aff1Ge[0  , 0] := 1.00000E+01; aff1Ge[0  , 1] := -2.69562E+01;
aff1Ge[1  , 0] := 1.99800E+01; aff1Ge[1  , 1] := -2.74605E+01;
aff1Ge[2  , 0] := 2.99600E+01; aff1Ge[2  , 1] := -2.88439E+01;
aff1Ge[3  , 0] := 3.99400E+01; aff1Ge[3  , 1] := -2.93110E+01;
aff1Ge[4  , 0] := 4.99200E+01; aff1Ge[4  , 1] := -2.98763E+01;
aff1Ge[5  , 0] := 5.99000E+01; aff1Ge[5  , 1] := -3.00073E+01;
aff1Ge[6  , 0] := 6.98800E+01; aff1Ge[6  , 1] := -2.96407E+01;
aff1Ge[7  , 0] := 7.98600E+01; aff1Ge[7  , 1] := -2.88592E+01;
aff1Ge[8  , 0] := 8.98400E+01; aff1Ge[8  , 1] := -2.77849E+01;
aff1Ge[9  , 0] := 9.98200E+01; aff1Ge[9  , 1] := -2.65823E+01;
aff1Ge[10 , 0] := 1.09800E+02; aff1Ge[10 , 1] := -2.53647E+01;
aff1Ge[11 , 0] := 1.19780E+02; aff1Ge[11 , 1] := -2.42993E+01;
aff1Ge[12 , 0] := 1.29760E+02; aff1Ge[12 , 1] := -2.30319E+01;
aff1Ge[13 , 0] := 1.39740E+02; aff1Ge[13 , 1] := -2.17280E+01;
aff1Ge[14 , 0] := 1.49720E+02; aff1Ge[14 , 1] := -2.05826E+01;
aff1Ge[15 , 0] := 1.59700E+02; aff1Ge[15 , 1] := -1.95740E+01;
aff1Ge[16 , 0] := 1.69680E+02; aff1Ge[16 , 1] := -1.87194E+01;
aff1Ge[17 , 0] := 1.79660E+02; aff1Ge[17 , 1] := -1.81208E+01;
aff1Ge[18 , 0] := 1.89640E+02; aff1Ge[18 , 1] := -1.70898E+01;
aff1Ge[19 , 0] := 1.99620E+02; aff1Ge[19 , 1] := -1.62563E+01;
aff1Ge[20 , 0] := 2.09600E+02; aff1Ge[20 , 1] := -1.55355E+01;
aff1Ge[21 , 0] := 2.19580E+02; aff1Ge[21 , 1] := -1.48945E+01;
aff1Ge[22 , 0] := 2.29560E+02; aff1Ge[22 , 1] := -1.43191E+01;
aff1Ge[23 , 0] := 2.39540E+02; aff1Ge[23 , 1] := -1.37997E+01;
aff1Ge[24 , 0] := 2.49520E+02; aff1Ge[24 , 1] := -1.33294E+01;
aff1Ge[25 , 0] := 2.59500E+02; aff1Ge[25 , 1] := -1.29022E+01;
aff1Ge[26 , 0] := 2.69480E+02; aff1Ge[26 , 1] := -1.25135E+01;
aff1Ge[27 , 0] := 2.79460E+02; aff1Ge[27 , 1] := -1.21589E+01;
aff1Ge[28 , 0] := 2.89440E+02; aff1Ge[28 , 1] := -1.18350E+01;
aff1Ge[29 , 0] := 2.99420E+02; aff1Ge[29 , 1] := -1.15386E+01;
aff1Ge[30 , 0] := 3.09400E+02; aff1Ge[30 , 1] := -1.12669E+01;
aff1Ge[31 , 0] := 3.19380E+02; aff1Ge[31 , 1] := -1.10176E+01;
aff1Ge[32 , 0] := 3.29360E+02; aff1Ge[32 , 1] := -1.07885E+01;
aff1Ge[33 , 0] := 3.39340E+02; aff1Ge[33 , 1] := -1.05777E+01;
aff1Ge[34 , 0] := 3.49320E+02; aff1Ge[34 , 1] := -1.03835E+01;
aff1Ge[35 , 0] := 3.59300E+02; aff1Ge[35 , 1] := -1.02046E+01;
aff1Ge[36 , 0] := 3.69280E+02; aff1Ge[36 , 1] := -1.00390E+01;
aff1Ge[37 , 0] := 3.79260E+02; aff1Ge[37 , 1] := -9.88636E+00;
aff1Ge[38 , 0] := 3.89240E+02; aff1Ge[38 , 1] := -9.74811E+00;
aff1Ge[39 , 0] := 3.99220E+02; aff1Ge[39 , 1] := -9.61794E+00;
aff1Ge[40 , 0] := 4.09200E+02; aff1Ge[40 , 1] := -9.49749E+00;
aff1Ge[41 , 0] := 4.19180E+02; aff1Ge[41 , 1] := -9.38606E+00;
aff1Ge[42 , 0] := 4.29160E+02; aff1Ge[42 , 1] := -9.28294E+00;
aff1Ge[43 , 0] := 4.39140E+02; aff1Ge[43 , 1] := -9.18748E+00;
aff1Ge[44 , 0] := 4.49120E+02; aff1Ge[44 , 1] := -9.09912E+00;
aff1Ge[45 , 0] := 4.59100E+02; aff1Ge[45 , 1] := -9.01731E+00;
aff1Ge[46 , 0] := 4.69080E+02; aff1Ge[46 , 1] := -8.94156E+00;
aff1Ge[47 , 0] := 4.79060E+02; aff1Ge[47 , 1] := -8.87141E+00;
aff1Ge[48 , 0] := 4.89040E+02; aff1Ge[48 , 1] := -8.80645E+00;
aff1Ge[49 , 0] := 4.99020E+02; aff1Ge[49 , 1] := -8.74631E+00;
aff1Ge[50 , 0] := 5.09000E+02; aff1Ge[50 , 1] := -8.69071E+00;
aff1Ge[51 , 0] := 5.18980E+02; aff1Ge[51 , 1] := -8.63934E+00;
aff1Ge[52 , 0] := 5.28960E+02; aff1Ge[52 , 1] := -8.59192E+00;
aff1Ge[53 , 0] := 5.38940E+02; aff1Ge[53 , 1] := -8.54809E+00;
aff1Ge[54 , 0] := 5.48920E+02; aff1Ge[54 , 1] := -8.50710E+00;
aff1Ge[55 , 0] := 5.58900E+02; aff1Ge[55 , 1] := -8.47410E+00;
aff1Ge[56 , 0] := 5.68880E+02; aff1Ge[56 , 1] := -8.44688E+00;
aff1Ge[57 , 0] := 5.78860E+02; aff1Ge[57 , 1] := -8.42499E+00;
aff1Ge[58 , 0] := 5.88840E+02; aff1Ge[58 , 1] := -8.40804E+00;
aff1Ge[59 , 0] := 5.98820E+02; aff1Ge[59 , 1] := -8.39568E+00;
aff1Ge[60 , 0] := 6.08800E+02; aff1Ge[60 , 1] := -8.38763E+00;
aff1Ge[61 , 0] := 6.18780E+02; aff1Ge[61 , 1] := -8.38361E+00;
aff1Ge[62 , 0] := 6.28760E+02; aff1Ge[62 , 1] := -8.38341E+00;
aff1Ge[63 , 0] := 6.38740E+02; aff1Ge[63 , 1] := -8.38682E+00;
aff1Ge[64 , 0] := 6.48720E+02; aff1Ge[64 , 1] := -8.39368E+00;
aff1Ge[65 , 0] := 6.58700E+02; aff1Ge[65 , 1] := -8.40382E+00;
aff1Ge[66 , 0] := 6.68680E+02; aff1Ge[66 , 1] := -8.41712E+00;
aff1Ge[67 , 0] := 6.78660E+02; aff1Ge[67 , 1] := -8.43346E+00;
aff1Ge[68 , 0] := 6.88640E+02; aff1Ge[68 , 1] := -8.45275E+00;
aff1Ge[69 , 0] := 6.98620E+02; aff1Ge[69 , 1] := -8.47490E+00;
aff1Ge[70 , 0] := 7.08600E+02; aff1Ge[70 , 1] := -8.49984E+00;
aff1Ge[71 , 0] := 7.18580E+02; aff1Ge[71 , 1] := -8.52752E+00;
aff1Ge[72 , 0] := 7.28560E+02; aff1Ge[72 , 1] := -8.55788E+00;
aff1Ge[73 , 0] := 7.38540E+02; aff1Ge[73 , 1] := -8.59091E+00;
aff1Ge[74 , 0] := 7.48520E+02; aff1Ge[74 , 1] := -8.62657E+00;
aff1Ge[75 , 0] := 7.58500E+02; aff1Ge[75 , 1] := -8.66487E+00;
aff1Ge[76 , 0] := 7.68480E+02; aff1Ge[76 , 1] := -8.70579E+00;
aff1Ge[77 , 0] := 7.78460E+02; aff1Ge[77 , 1] := -8.74937E+00;
aff1Ge[78 , 0] := 7.88440E+02; aff1Ge[78 , 1] := -8.79560E+00;
aff1Ge[79 , 0] := 7.98420E+02; aff1Ge[79 , 1] := -8.84453E+00;
aff1Ge[80 , 0] := 8.08400E+02; aff1Ge[80 , 1] := -8.89620E+00;
aff1Ge[81 , 0] := 8.18380E+02; aff1Ge[81 , 1] := -8.95066E+00;
aff1Ge[82 , 0] := 8.28360E+02; aff1Ge[82 , 1] := -9.00798E+00;
aff1Ge[83 , 0] := 8.38340E+02; aff1Ge[83 , 1] := -9.06823E+00;
aff1Ge[84 , 0] := 8.48320E+02; aff1Ge[84 , 1] := -9.13150E+00;
aff1Ge[85 , 0] := 8.58300E+02; aff1Ge[85 , 1] := -9.19789E+00;
aff1Ge[86 , 0] := 8.68280E+02; aff1Ge[86 , 1] := -9.26753E+00;
aff1Ge[87 , 0] := 8.78260E+02; aff1Ge[87 , 1] := -9.34054E+00;
aff1Ge[88 , 0] := 8.88240E+02; aff1Ge[88 , 1] := -9.41707E+00;
aff1Ge[89 , 0] := 8.98220E+02; aff1Ge[89 , 1] := -9.49731E+00;
aff1Ge[90 , 0] := 9.08200E+02; aff1Ge[90 , 1] := -9.58142E+00;
aff1Ge[91 , 0] := 9.18180E+02; aff1Ge[91 , 1] := -9.66964E+00;
aff1Ge[92 , 0] := 9.28160E+02; aff1Ge[92 , 1] := -9.76220E+00;
aff1Ge[93 , 0] := 9.38140E+02; aff1Ge[93 , 1] := -9.85936E+00;
aff1Ge[94 , 0] := 9.48120E+02; aff1Ge[94 , 1] := -9.96144E+00;
aff1Ge[95 , 0] := 9.58100E+02; aff1Ge[95 , 1] := -1.00688E+01;
aff1Ge[96 , 0] := 9.68080E+02; aff1Ge[96 , 1] := -1.01817E+01;
aff1Ge[97 , 0] := 9.78060E+02; aff1Ge[97 , 1] := -1.03008E+01;
aff1Ge[98 , 0] := 9.88040E+02; aff1Ge[98 , 1] := -1.04264E+01;
aff1Ge[99 , 0] := 9.98020E+02; aff1Ge[99 , 1] := -1.05588E+01;
aff1Ge[100, 0] := 1.00800E+03; aff1Ge[100, 1] := -1.06740E+01;
aff1Ge[101, 0] := 1.01798E+03; aff1Ge[101, 1] := -1.08082E+01;
aff1Ge[102, 0] := 1.02796E+03; aff1Ge[102, 1] := -1.09580E+01;
aff1Ge[103, 0] := 1.03794E+03; aff1Ge[103, 1] := -1.11214E+01;
aff1Ge[104, 0] := 1.04792E+03; aff1Ge[104, 1] := -1.12984E+01;
aff1Ge[105, 0] := 1.05790E+03; aff1Ge[105, 1] := -1.14900E+01;
aff1Ge[106, 0] := 1.06788E+03; aff1Ge[106, 1] := -1.16973E+01;
aff1Ge[107, 0] := 1.07786E+03; aff1Ge[107, 1] := -1.19223E+01;
aff1Ge[108, 0] := 1.08784E+03; aff1Ge[108, 1] := -1.21671E+01;
aff1Ge[109, 0] := 1.09782E+03; aff1Ge[109, 1] := -1.24347E+01;
aff1Ge[110, 0] := 1.10780E+03; aff1Ge[110, 1] := -1.27288E+01;
aff1Ge[111, 0] := 1.11778E+03; aff1Ge[111, 1] := -1.30542E+01;
aff1Ge[112, 0] := 1.12776E+03; aff1Ge[112, 1] := -1.34172E+01;
aff1Ge[113, 0] := 1.13774E+03; aff1Ge[113, 1] := -1.38264E+01;
aff1Ge[114, 0] := 1.14772E+03; aff1Ge[114, 1] := -1.42937E+01;
aff1Ge[115, 0] := 1.15770E+03; aff1Ge[115, 1] := -1.48367E+01;
aff1Ge[116, 0] := 1.16768E+03; aff1Ge[116, 1] := -1.54822E+01;
aff1Ge[117, 0] := 1.17766E+03; aff1Ge[117, 1] := -1.62764E+01;
aff1Ge[118, 0] := 1.18764E+03; aff1Ge[118, 1] := -1.73070E+01;
aff1Ge[119, 0] := 1.19762E+03; aff1Ge[119, 1] := -1.87288E+01;
aff1Ge[120, 0] := 1.20760E+03; aff1Ge[120, 1] := -2.12100E+01;
aff1Ge[121, 0] := 1.21758E+03; aff1Ge[121, 1] := -2.83958E+01;
aff1Ge[122, 0] := 1.22756E+03; aff1Ge[122, 1] := -2.14204E+01;
aff1Ge[123, 0] := 1.23754E+03; aff1Ge[123, 1] := -2.02584E+01;
aff1Ge[124, 0] := 1.24752E+03; aff1Ge[124, 1] := -2.36131E+01;
aff1Ge[125, 0] := 1.25750E+03; aff1Ge[125, 1] := -1.80663E+01;
aff1Ge[126, 0] := 1.26748E+03; aff1Ge[126, 1] := -1.62455E+01;
aff1Ge[127, 0] := 1.27746E+03; aff1Ge[127, 1] := -1.49931E+01;
aff1Ge[128, 0] := 1.28744E+03; aff1Ge[128, 1] := -1.40188E+01;
aff1Ge[129, 0] := 1.29742E+03; aff1Ge[129, 1] := -1.32303E+01;
aff1Ge[130, 0] := 1.30740E+03; aff1Ge[130, 1] := -1.25660E+01;
aff1Ge[131, 0] := 1.31738E+03; aff1Ge[131, 1] := -1.19953E+01;
aff1Ge[132, 0] := 1.32736E+03; aff1Ge[132, 1] := -1.15004E+01;
aff1Ge[133, 0] := 1.33734E+03; aff1Ge[133, 1] := -1.10692E+01;
aff1Ge[134, 0] := 1.34732E+03; aff1Ge[134, 1] := -1.06941E+01;
aff1Ge[135, 0] := 1.35730E+03; aff1Ge[135, 1] := -1.03708E+01;
aff1Ge[136, 0] := 1.36728E+03; aff1Ge[136, 1] := -1.00987E+01;
aff1Ge[137, 0] := 1.37726E+03; aff1Ge[137, 1] := -9.88117E+00;
aff1Ge[138, 0] := 1.38724E+03; aff1Ge[138, 1] := -9.72484E+00;
aff1Ge[139, 0] := 1.39722E+03; aff1Ge[139, 1] := -9.66231E+00;
aff1Ge[140, 0] := 1.40720E+03; aff1Ge[140, 1] := -9.90064E+00;
aff1Ge[141, 0] := 1.41718E+03; aff1Ge[141, 1] := -9.89144E+00;
aff1Ge[142, 0] := 1.42716E+03; aff1Ge[142, 1] := -9.04354E+00;
aff1Ge[143, 0] := 1.43714E+03; aff1Ge[143, 1] := -8.44440E+00;
aff1Ge[144, 0] := 1.44712E+03; aff1Ge[144, 1] := -8.04837E+00;
aff1Ge[145, 0] := 1.45710E+03; aff1Ge[145, 1] := -7.66433E+00;
aff1Ge[146, 0] := 1.46708E+03; aff1Ge[146, 1] := -7.33565E+00;
aff1Ge[147, 0] := 1.47706E+03; aff1Ge[147, 1] := -7.03836E+00;
aff1Ge[148, 0] := 1.48704E+03; aff1Ge[148, 1] := -6.76578E+00;
aff1Ge[149, 0] := 1.49702E+03; aff1Ge[149, 1] := -6.51318E+00;
aff1Ge[150, 0] := 1.50700E+03; aff1Ge[150, 1] := -6.27757E+00;
aff1Ge[151, 0] := 1.51698E+03; aff1Ge[151, 1] := -6.05663E+00;
aff1Ge[152, 0] := 1.52696E+03; aff1Ge[152, 1] := -5.84846E+00;
aff1Ge[153, 0] := 1.53694E+03; aff1Ge[153, 1] := -5.65164E+00;
aff1Ge[154, 0] := 1.54692E+03; aff1Ge[154, 1] := -5.46502E+00;
aff1Ge[155, 0] := 1.55690E+03; aff1Ge[155, 1] := -5.28758E+00;
aff1Ge[156, 0] := 1.56688E+03; aff1Ge[156, 1] := -5.11849E+00;
aff1Ge[157, 0] := 1.57686E+03; aff1Ge[157, 1] := -4.95701E+00;
aff1Ge[158, 0] := 1.58684E+03; aff1Ge[158, 1] := -4.80260E+00;
aff1Ge[159, 0] := 1.59682E+03; aff1Ge[159, 1] := -4.65490E+00;
aff1Ge[160, 0] := 1.60680E+03; aff1Ge[160, 1] := -4.51353E+00;
aff1Ge[161, 0] := 1.61678E+03; aff1Ge[161, 1] := -4.37793E+00;
aff1Ge[162, 0] := 1.62676E+03; aff1Ge[162, 1] := -4.24779E+00;
aff1Ge[163, 0] := 1.63674E+03; aff1Ge[163, 1] := -4.12289E+00;
aff1Ge[164, 0] := 1.64672E+03; aff1Ge[164, 1] := -4.00290E+00;
aff1Ge[165, 0] := 1.65670E+03; aff1Ge[165, 1] := -3.88754E+00;
aff1Ge[166, 0] := 1.66668E+03; aff1Ge[166, 1] := -3.77652E+00;
aff1Ge[167, 0] := 1.67666E+03; aff1Ge[167, 1] := -3.66960E+00;
aff1Ge[168, 0] := 1.68664E+03; aff1Ge[168, 1] := -3.56654E+00;
aff1Ge[169, 0] := 1.69662E+03; aff1Ge[169, 1] := -3.46715E+00;
aff1Ge[170, 0] := 1.70660E+03; aff1Ge[170, 1] := -3.37123E+00;
aff1Ge[171, 0] := 1.71658E+03; aff1Ge[171, 1] := -3.27860E+00;
aff1Ge[172, 0] := 1.72656E+03; aff1Ge[172, 1] := -3.18910E+00;
aff1Ge[173, 0] := 1.73654E+03; aff1Ge[173, 1] := -3.10258E+00;
aff1Ge[174, 0] := 1.74652E+03; aff1Ge[174, 1] := -3.01889E+00;
aff1Ge[175, 0] := 1.75650E+03; aff1Ge[175, 1] := -2.93789E+00;
aff1Ge[176, 0] := 1.76648E+03; aff1Ge[176, 1] := -2.85946E+00;
aff1Ge[177, 0] := 1.77646E+03; aff1Ge[177, 1] := -2.78347E+00;
aff1Ge[178, 0] := 1.78644E+03; aff1Ge[178, 1] := -2.70981E+00;
aff1Ge[179, 0] := 1.79642E+03; aff1Ge[179, 1] := -2.63837E+00;
aff1Ge[180, 0] := 1.80640E+03; aff1Ge[180, 1] := -2.56904E+00;
aff1Ge[181, 0] := 1.81638E+03; aff1Ge[181, 1] := -2.50168E+00;
aff1Ge[182, 0] := 1.82636E+03; aff1Ge[182, 1] := -2.43620E+00;
aff1Ge[183, 0] := 1.83634E+03; aff1Ge[183, 1] := -2.37250E+00;
aff1Ge[184, 0] := 1.84632E+03; aff1Ge[184, 1] := -2.31060E+00;
aff1Ge[185, 0] := 1.85630E+03; aff1Ge[185, 1] := -2.25066E+00;
aff1Ge[186, 0] := 1.86628E+03; aff1Ge[186, 1] := -2.19265E+00;
aff1Ge[187, 0] := 1.87626E+03; aff1Ge[187, 1] := -2.13640E+00;
aff1Ge[188, 0] := 1.88624E+03; aff1Ge[188, 1] := -2.08183E+00;
aff1Ge[189, 0] := 1.89622E+03; aff1Ge[189, 1] := -2.02888E+00;
aff1Ge[190, 0] := 1.90620E+03; aff1Ge[190, 1] := -1.97748E+00;
aff1Ge[191, 0] := 1.91618E+03; aff1Ge[191, 1] := -1.92757E+00;
aff1Ge[192, 0] := 1.92616E+03; aff1Ge[192, 1] := -1.87908E+00;
aff1Ge[193, 0] := 1.93614E+03; aff1Ge[193, 1] := -1.83197E+00;
aff1Ge[194, 0] := 1.94612E+03; aff1Ge[194, 1] := -1.78618E+00;
aff1Ge[195, 0] := 1.95610E+03; aff1Ge[195, 1] := -1.74166E+00;
aff1Ge[196, 0] := 1.96608E+03; aff1Ge[196, 1] := -1.69837E+00;
aff1Ge[197, 0] := 1.97606E+03; aff1Ge[197, 1] := -1.65627E+00;
aff1Ge[198, 0] := 1.98604E+03; aff1Ge[198, 1] := -1.61531E+00;
aff1Ge[199, 0] := 1.99602E+03; aff1Ge[199, 1] := -1.57545E+00;
aff1Ge[200, 0] := 2.00600E+03; aff1Ge[200, 1] := -1.53666E+00;
aff1Ge[201, 0] := 2.01598E+03; aff1Ge[201, 1] := -1.49890E+00;
aff1Ge[202, 0] := 2.02596E+03; aff1Ge[202, 1] := -1.46214E+00;
aff1Ge[203, 0] := 2.03594E+03; aff1Ge[203, 1] := -1.42634E+00;
aff1Ge[204, 0] := 2.04592E+03; aff1Ge[204, 1] := -1.39147E+00;
aff1Ge[205, 0] := 2.05590E+03; aff1Ge[205, 1] := -1.35750E+00;
aff1Ge[206, 0] := 2.06588E+03; aff1Ge[206, 1] := -1.32440E+00;
aff1Ge[207, 0] := 2.07586E+03; aff1Ge[207, 1] := -1.29215E+00;
aff1Ge[208, 0] := 2.08584E+03; aff1Ge[208, 1] := -1.26072E+00;
aff1Ge[209, 0] := 2.09582E+03; aff1Ge[209, 1] := -1.23008E+00;
aff1Ge[210, 0] := 2.10580E+03; aff1Ge[210, 1] := -1.20020E+00;
aff1Ge[211, 0] := 2.11578E+03; aff1Ge[211, 1] := -1.17107E+00;
aff1Ge[212, 0] := 2.12576E+03; aff1Ge[212, 1] := -1.14266E+00;
aff1Ge[213, 0] := 2.13574E+03; aff1Ge[213, 1] := -1.11495E+00;
aff1Ge[214, 0] := 2.14572E+03; aff1Ge[214, 1] := -1.08791E+00;
aff1Ge[215, 0] := 2.15570E+03; aff1Ge[215, 1] := -1.06153E+00;
aff1Ge[216, 0] := 2.16568E+03; aff1Ge[216, 1] := -1.03578E+00;
aff1Ge[217, 0] := 2.17566E+03; aff1Ge[217, 1] := -1.01065E+00;
aff1Ge[218, 0] := 2.18564E+03; aff1Ge[218, 1] := -9.86115E-01;
aff1Ge[219, 0] := 2.19562E+03; aff1Ge[219, 1] := -9.62161E-01;
aff1Ge[220, 0] := 2.20560E+03; aff1Ge[220, 1] := -9.38768E-01;
aff1Ge[221, 0] := 2.21558E+03; aff1Ge[221, 1] := -9.15920E-01;
aff1Ge[222, 0] := 2.22556E+03; aff1Ge[222, 1] := -8.93600E-01;
aff1Ge[223, 0] := 2.23554E+03; aff1Ge[223, 1] := -8.71792E-01;
aff1Ge[224, 0] := 2.24552E+03; aff1Ge[224, 1] := -8.50481E-01;
aff1Ge[225, 0] := 2.25550E+03; aff1Ge[225, 1] := -8.29650E-01;
aff1Ge[226, 0] := 2.26548E+03; aff1Ge[226, 1] := -8.09280E-01;
aff1Ge[227, 0] := 2.27546E+03; aff1Ge[227, 1] := -7.89365E-01;
aff1Ge[228, 0] := 2.28544E+03; aff1Ge[228, 1] := -7.69901E-01;
aff1Ge[229, 0] := 2.29542E+03; aff1Ge[229, 1] := -7.50878E-01;
aff1Ge[230, 0] := 2.30540E+03; aff1Ge[230, 1] := -7.32285E-01;
aff1Ge[231, 0] := 2.31538E+03; aff1Ge[231, 1] := -7.14109E-01;
aff1Ge[232, 0] := 2.32536E+03; aff1Ge[232, 1] := -6.96337E-01;
aff1Ge[233, 0] := 2.33534E+03; aff1Ge[233, 1] := -6.78955E-01;
aff1Ge[234, 0] := 2.34532E+03; aff1Ge[234, 1] := -6.61952E-01;
aff1Ge[235, 0] := 2.35530E+03; aff1Ge[235, 1] := -6.45314E-01;
aff1Ge[236, 0] := 2.36528E+03; aff1Ge[236, 1] := -6.29029E-01;
aff1Ge[237, 0] := 2.37526E+03; aff1Ge[237, 1] := -6.12652E-01;
aff1Ge[238, 0] := 2.38524E+03; aff1Ge[238, 1] := -5.96113E-01;
aff1Ge[239, 0] := 2.39522E+03; aff1Ge[239, 1] := -5.82297E-01;
aff1Ge[240, 0] := 2.40520E+03; aff1Ge[240, 1] := -5.75274E-01;
aff1Ge[241, 0] := 2.41518E+03; aff1Ge[241, 1] := -5.59237E-01;
aff1Ge[242, 0] := 2.42516E+03; aff1Ge[242, 1] := -5.14714E-01;
aff1Ge[243, 0] := 2.43514E+03; aff1Ge[243, 1] := -4.50058E-01;
aff1Ge[244, 0] := 2.44512E+03; aff1Ge[244, 1] := -3.97799E-01;
aff1Ge[245, 0] := 2.45510E+03; aff1Ge[245, 1] := -3.77479E-01;
aff1Ge[246, 0] := 2.46508E+03; aff1Ge[246, 1] := -3.73610E-01;
aff1Ge[247, 0] := 2.47506E+03; aff1Ge[247, 1] := -3.69250E-01;
aff1Ge[248, 0] := 2.48504E+03; aff1Ge[248, 1] := -3.57644E-01;
aff1Ge[249, 0] := 2.49502E+03; aff1Ge[249, 1] := -3.34697E-01;
aff1Ge[250, 0] := 2.50500E+03; aff1Ge[250, 1] := -2.99806E-01;
aff1Ge[251, 0] := 2.51498E+03; aff1Ge[251, 1] := -2.65560E-01;
aff1Ge[252, 0] := 2.52496E+03; aff1Ge[252, 1] := -2.45184E-01;
aff1Ge[253, 0] := 2.53494E+03; aff1Ge[253, 1] := -2.36730E-01;
aff1Ge[254, 0] := 2.54492E+03; aff1Ge[254, 1] := -2.30689E-01;
aff1Ge[255, 0] := 2.55490E+03; aff1Ge[255, 1] := -2.21323E-01;
aff1Ge[256, 0] := 2.56488E+03; aff1Ge[256, 1] := -2.10582E-01;
aff1Ge[257, 0] := 2.57486E+03; aff1Ge[257, 1] := -2.00644E-01;
aff1Ge[258, 0] := 2.58484E+03; aff1Ge[258, 1] := -1.91524E-01;
aff1Ge[259, 0] := 2.59482E+03; aff1Ge[259, 1] := -1.82754E-01;
aff1Ge[260, 0] := 2.60480E+03; aff1Ge[260, 1] := -1.74093E-01;
aff1Ge[261, 0] := 2.61478E+03; aff1Ge[261, 1] := -1.65674E-01;
aff1Ge[262, 0] := 2.62476E+03; aff1Ge[262, 1] := -1.57485E-01;
aff1Ge[263, 0] := 2.63474E+03; aff1Ge[263, 1] := -1.49519E-01;
aff1Ge[264, 0] := 2.64472E+03; aff1Ge[264, 1] := -1.41769E-01;
aff1Ge[265, 0] := 2.65470E+03; aff1Ge[265, 1] := -1.34226E-01;
aff1Ge[266, 0] := 2.66468E+03; aff1Ge[266, 1] := -1.26883E-01;
aff1Ge[267, 0] := 2.67466E+03; aff1Ge[267, 1] := -1.19734E-01;
aff1Ge[268, 0] := 2.68464E+03; aff1Ge[268, 1] := -1.12771E-01;
aff1Ge[269, 0] := 2.69462E+03; aff1Ge[269, 1] := -1.05986E-01;
aff1Ge[270, 0] := 2.70460E+03; aff1Ge[270, 1] := -9.93742E-02;
aff1Ge[271, 0] := 2.71458E+03; aff1Ge[271, 1] := -9.29281E-02;
aff1Ge[272, 0] := 2.72456E+03; aff1Ge[272, 1] := -8.66415E-02;
aff1Ge[273, 0] := 2.73454E+03; aff1Ge[273, 1] := -8.05081E-02;
aff1Ge[274, 0] := 2.74452E+03; aff1Ge[274, 1] := -7.45217E-02;
aff1Ge[275, 0] := 2.75450E+03; aff1Ge[275, 1] := -6.86282E-02;
aff1Ge[276, 0] := 2.76448E+03; aff1Ge[276, 1] := -6.25366E-02;
aff1Ge[277, 0] := 2.77446E+03; aff1Ge[277, 1] := -5.69380E-02;
aff1Ge[278, 0] := 2.78444E+03; aff1Ge[278, 1] := -5.28992E-02;
aff1Ge[279, 0] := 2.79442E+03; aff1Ge[279, 1] := -5.00507E-02;
aff1Ge[280, 0] := 2.80440E+03; aff1Ge[280, 1] := -4.37488E-02;
aff1Ge[281, 0] := 2.81438E+03; aff1Ge[281, 1] := -2.89914E-02;
aff1Ge[282, 0] := 2.82436E+03; aff1Ge[282, 1] := -7.54646E-03;
aff1Ge[283, 0] := 2.83434E+03; aff1Ge[283, 1] := 1.26428E-02;
aff1Ge[284, 0] := 2.84432E+03; aff1Ge[284, 1] := 2.41131E-02;
aff1Ge[285, 0] := 2.85430E+03; aff1Ge[285, 1] := 2.81389E-02;
aff1Ge[286, 0] := 2.86428E+03; aff1Ge[286, 1] := 2.97028E-02;
aff1Ge[287, 0] := 2.87426E+03; aff1Ge[287, 1] := 3.31872E-02;
aff1Ge[288, 0] := 2.88424E+03; aff1Ge[288, 1] := 3.81167E-02;
aff1Ge[289, 0] := 2.89422E+03; aff1Ge[289, 1] := 4.33388E-02;
aff1Ge[290, 0] := 2.90420E+03; aff1Ge[290, 1] := 4.79083E-02;
aff1Ge[291, 0] := 2.91418E+03; aff1Ge[291, 1] := 5.22285E-02;
aff1Ge[292, 0] := 2.92416E+03; aff1Ge[292, 1] := 5.64816E-02;
aff1Ge[293, 0] := 2.93414E+03; aff1Ge[293, 1] := 6.07854E-02;
aff1Ge[294, 0] := 2.94412E+03; aff1Ge[294, 1] := 6.50841E-02;
aff1Ge[295, 0] := 2.95410E+03; aff1Ge[295, 1] := 6.94052E-02;
aff1Ge[296, 0] := 2.96408E+03; aff1Ge[296, 1] := 7.37453E-02;
aff1Ge[297, 0] := 2.97406E+03; aff1Ge[297, 1] := 7.80791E-02;
aff1Ge[298, 0] := 2.98404E+03; aff1Ge[298, 1] := 8.23847E-02;
aff1Ge[299, 0] := 2.99402E+03; aff1Ge[299, 1] := 8.66198E-02;
aff1Ge[300, 0] := 3.00400E+03; aff1Ge[300, 1] := 9.05836E-02;
aff1Ge[301, 0] := 3.01398E+03; aff1Ge[301, 1] := 9.40748E-02;
aff1Ge[302, 0] := 3.02396E+03; aff1Ge[302, 1] := 9.70019E-02;
aff1Ge[303, 0] := 3.03394E+03; aff1Ge[303, 1] := 9.95317E-02;
aff1Ge[304, 0] := 3.04392E+03; aff1Ge[304, 1] := 1.01846E-01;
aff1Ge[305, 0] := 3.05390E+03; aff1Ge[305, 1] := 1.04055E-01;
aff1Ge[306, 0] := 3.06388E+03; aff1Ge[306, 1] := 1.06132E-01;
aff1Ge[307, 0] := 3.07386E+03; aff1Ge[307, 1] := 1.08041E-01;
aff1Ge[308, 0] := 3.08384E+03; aff1Ge[308, 1] := 1.09764E-01;
aff1Ge[309, 0] := 3.09382E+03; aff1Ge[309, 1] := 1.11324E-01;
aff1Ge[310, 0] := 3.10380E+03; aff1Ge[310, 1] := 1.12734E-01;
aff1Ge[311, 0] := 3.11378E+03; aff1Ge[311, 1] := 1.14006E-01;
aff1Ge[312, 0] := 3.12376E+03; aff1Ge[312, 1] := 1.15140E-01;
aff1Ge[313, 0] := 3.13374E+03; aff1Ge[313, 1] := 1.16144E-01;
aff1Ge[314, 0] := 3.14372E+03; aff1Ge[314, 1] := 1.17021E-01;
aff1Ge[315, 0] := 3.15370E+03; aff1Ge[315, 1] := 1.17778E-01;
aff1Ge[316, 0] := 3.16368E+03; aff1Ge[316, 1] := 1.18418E-01;
aff1Ge[317, 0] := 3.17366E+03; aff1Ge[317, 1] := 1.18946E-01;
aff1Ge[318, 0] := 3.18364E+03; aff1Ge[318, 1] := 1.19366E-01;
aff1Ge[319, 0] := 3.19362E+03; aff1Ge[319, 1] := 1.19682E-01;
aff1Ge[320, 0] := 3.20360E+03; aff1Ge[320, 1] := 1.19898E-01;
aff1Ge[321, 0] := 3.21358E+03; aff1Ge[321, 1] := 1.20018E-01;
aff1Ge[322, 0] := 3.22356E+03; aff1Ge[322, 1] := 1.20044E-01;
aff1Ge[323, 0] := 3.23354E+03; aff1Ge[323, 1] := 1.19980E-01;
aff1Ge[324, 0] := 3.24352E+03; aff1Ge[324, 1] := 1.19829E-01;
aff1Ge[325, 0] := 3.25350E+03; aff1Ge[325, 1] := 1.19594E-01;
aff1Ge[326, 0] := 3.26348E+03; aff1Ge[326, 1] := 1.19278E-01;
aff1Ge[327, 0] := 3.27346E+03; aff1Ge[327, 1] := 1.18883E-01;
aff1Ge[328, 0] := 3.28344E+03; aff1Ge[328, 1] := 1.18412E-01;
aff1Ge[329, 0] := 3.29342E+03; aff1Ge[329, 1] := 1.17868E-01;
aff1Ge[330, 0] := 3.30340E+03; aff1Ge[330, 1] := 1.17252E-01;
aff1Ge[331, 0] := 3.31338E+03; aff1Ge[331, 1] := 1.16567E-01;
aff1Ge[332, 0] := 3.32336E+03; aff1Ge[332, 1] := 1.15815E-01;
aff1Ge[333, 0] := 3.33334E+03; aff1Ge[333, 1] := 1.14999E-01;
aff1Ge[334, 0] := 3.34332E+03; aff1Ge[334, 1] := 1.14120E-01;
aff1Ge[335, 0] := 3.35330E+03; aff1Ge[335, 1] := 1.13181E-01;
aff1Ge[336, 0] := 3.36328E+03; aff1Ge[336, 1] := 1.12183E-01;
aff1Ge[337, 0] := 3.37326E+03; aff1Ge[337, 1] := 1.11128E-01;
aff1Ge[338, 0] := 3.38324E+03; aff1Ge[338, 1] := 1.10018E-01;
aff1Ge[339, 0] := 3.39322E+03; aff1Ge[339, 1] := 1.08854E-01;
aff1Ge[340, 0] := 3.40320E+03; aff1Ge[340, 1] := 1.07637E-01;
aff1Ge[341, 0] := 3.41318E+03; aff1Ge[341, 1] := 1.06368E-01;
aff1Ge[342, 0] := 3.42316E+03; aff1Ge[342, 1] := 1.05048E-01;
aff1Ge[343, 0] := 3.43314E+03; aff1Ge[343, 1] := 1.03679E-01;
aff1Ge[344, 0] := 3.44312E+03; aff1Ge[344, 1] := 1.02262E-01;
aff1Ge[345, 0] := 3.45310E+03; aff1Ge[345, 1] := 1.00799E-01;
aff1Ge[346, 0] := 3.46308E+03; aff1Ge[346, 1] := 9.92909E-02;
aff1Ge[347, 0] := 3.47306E+03; aff1Ge[347, 1] := 9.77392E-02;
aff1Ge[348, 0] := 3.48304E+03; aff1Ge[348, 1] := 9.61452E-02;
aff1Ge[349, 0] := 3.49302E+03; aff1Ge[349, 1] := 9.45101E-02;
aff1Ge[350, 0] := 3.50300E+03; aff1Ge[350, 1] := 9.28352E-02;
aff1Ge[351, 0] := 3.51298E+03; aff1Ge[351, 1] := 9.11215E-02;
aff1Ge[352, 0] := 3.52296E+03; aff1Ge[352, 1] := 8.93701E-02;
aff1Ge[353, 0] := 3.53294E+03; aff1Ge[353, 1] := 8.75824E-02;
aff1Ge[354, 0] := 3.54292E+03; aff1Ge[354, 1] := 8.57592E-02;
aff1Ge[355, 0] := 3.55290E+03; aff1Ge[355, 1] := 8.39017E-02;
aff1Ge[356, 0] := 3.56288E+03; aff1Ge[356, 1] := 8.20109E-02;
aff1Ge[357, 0] := 3.57286E+03; aff1Ge[357, 1] := 8.00876E-02;
aff1Ge[358, 0] := 3.58284E+03; aff1Ge[358, 1] := 7.81329E-02;
aff1Ge[359, 0] := 3.59282E+03; aff1Ge[359, 1] := 7.61477E-02;
aff1Ge[360, 0] := 3.60280E+03; aff1Ge[360, 1] := 7.41329E-02;
aff1Ge[361, 0] := 3.61278E+03; aff1Ge[361, 1] := 7.20894E-02;
aff1Ge[362, 0] := 3.62276E+03; aff1Ge[362, 1] := 7.00180E-02;
aff1Ge[363, 0] := 3.63274E+03; aff1Ge[363, 1] := 6.79195E-02;
aff1Ge[364, 0] := 3.64272E+03; aff1Ge[364, 1] := 6.57948E-02;
aff1Ge[365, 0] := 3.65270E+03; aff1Ge[365, 1] := 6.36446E-02;
aff1Ge[366, 0] := 3.66268E+03; aff1Ge[366, 1] := 6.14697E-02;
aff1Ge[367, 0] := 3.67266E+03; aff1Ge[367, 1] := 5.92708E-02;
aff1Ge[368, 0] := 3.68264E+03; aff1Ge[368, 1] := 5.70486E-02;
aff1Ge[369, 0] := 3.69262E+03; aff1Ge[369, 1] := 5.48039E-02;
aff1Ge[370, 0] := 3.70260E+03; aff1Ge[370, 1] := 5.25373E-02;
aff1Ge[371, 0] := 3.71258E+03; aff1Ge[371, 1] := 5.02496E-02;
aff1Ge[372, 0] := 3.72256E+03; aff1Ge[372, 1] := 4.79412E-02;
aff1Ge[373, 0] := 3.73254E+03; aff1Ge[373, 1] := 4.56129E-02;
aff1Ge[374, 0] := 3.74252E+03; aff1Ge[374, 1] := 4.32653E-02;
aff1Ge[375, 0] := 3.75250E+03; aff1Ge[375, 1] := 4.08990E-02;
aff1Ge[376, 0] := 3.76248E+03; aff1Ge[376, 1] := 3.85145E-02;
aff1Ge[377, 0] := 3.77246E+03; aff1Ge[377, 1] := 3.61125E-02;
aff1Ge[378, 0] := 3.78244E+03; aff1Ge[378, 1] := 3.36934E-02;
aff1Ge[379, 0] := 3.79242E+03; aff1Ge[379, 1] := 3.12578E-02;
aff1Ge[380, 0] := 3.80240E+03; aff1Ge[380, 1] := 2.88062E-02;
aff1Ge[381, 0] := 3.81238E+03; aff1Ge[381, 1] := 2.63392E-02;
aff1Ge[382, 0] := 3.82236E+03; aff1Ge[382, 1] := 2.38572E-02;
aff1Ge[383, 0] := 3.83234E+03; aff1Ge[383, 1] := 2.13608E-02;
aff1Ge[384, 0] := 3.84232E+03; aff1Ge[384, 1] := 1.88503E-02;
aff1Ge[385, 0] := 3.85230E+03; aff1Ge[385, 1] := 1.63263E-02;
aff1Ge[386, 0] := 3.86228E+03; aff1Ge[386, 1] := 1.37892E-02;
aff1Ge[387, 0] := 3.87226E+03; aff1Ge[387, 1] := 1.12394E-02;
aff1Ge[388, 0] := 3.88224E+03; aff1Ge[388, 1] := 8.67742E-03;
aff1Ge[389, 0] := 3.89222E+03; aff1Ge[389, 1] := 6.10361E-03;
aff1Ge[390, 0] := 3.90220E+03; aff1Ge[390, 1] := 3.51839E-03;
aff1Ge[391, 0] := 3.91218E+03; aff1Ge[391, 1] := 9.22167E-04;
aff1Ge[392, 0] := 3.92216E+03; aff1Ge[392, 1] := -1.68468E-03;
aff1Ge[393, 0] := 3.93214E+03; aff1Ge[393, 1] := -4.30178E-03;
aff1Ge[394, 0] := 3.94212E+03; aff1Ge[394, 1] := -6.92875E-03;
aff1Ge[395, 0] := 3.95210E+03; aff1Ge[395, 1] := -9.56523E-03;
aff1Ge[396, 0] := 3.96208E+03; aff1Ge[396, 1] := -1.22109E-02;
aff1Ge[397, 0] := 3.97206E+03; aff1Ge[397, 1] := -1.48653E-02;
aff1Ge[398, 0] := 3.98204E+03; aff1Ge[398, 1] := -1.75283E-02;
aff1Ge[399, 0] := 3.99202E+03; aff1Ge[399, 1] := -2.01994E-02;
aff1Ge[400, 0] := 4.00200E+03; aff1Ge[400, 1] := -2.28784E-02;
aff1Ge[401, 0] := 4.01198E+03; aff1Ge[401, 1] := -2.55650E-02;
aff1Ge[402, 0] := 4.02196E+03; aff1Ge[402, 1] := -2.82587E-02;
aff1Ge[403, 0] := 4.03194E+03; aff1Ge[403, 1] := -3.09595E-02;
aff1Ge[404, 0] := 4.04192E+03; aff1Ge[404, 1] := -3.36668E-02;
aff1Ge[405, 0] := 4.05190E+03; aff1Ge[405, 1] := -3.63806E-02;
aff1Ge[406, 0] := 4.06188E+03; aff1Ge[406, 1] := -3.91005E-02;
aff1Ge[407, 0] := 4.07186E+03; aff1Ge[407, 1] := -4.18261E-02;
aff1Ge[408, 0] := 4.08184E+03; aff1Ge[408, 1] := -4.45573E-02;
aff1Ge[409, 0] := 4.09182E+03; aff1Ge[409, 1] := -4.72939E-02;
aff1Ge[410, 0] := 4.10180E+03; aff1Ge[410, 1] := -5.00355E-02;
aff1Ge[411, 0] := 4.11178E+03; aff1Ge[411, 1] := -5.27820E-02;
aff1Ge[412, 0] := 4.12176E+03; aff1Ge[412, 1] := -5.55330E-02;
aff1Ge[413, 0] := 4.13174E+03; aff1Ge[413, 1] := -5.82884E-02;
aff1Ge[414, 0] := 4.14172E+03; aff1Ge[414, 1] := -6.10479E-02;
aff1Ge[415, 0] := 4.15170E+03; aff1Ge[415, 1] := -6.38113E-02;
aff1Ge[416, 0] := 4.16168E+03; aff1Ge[416, 1] := -6.65784E-02;
aff1Ge[417, 0] := 4.17166E+03; aff1Ge[417, 1] := -6.93490E-02;
aff1Ge[418, 0] := 4.18164E+03; aff1Ge[418, 1] := -7.21229E-02;
aff1Ge[419, 0] := 4.19162E+03; aff1Ge[419, 1] := -7.48998E-02;
aff1Ge[420, 0] := 4.20160E+03; aff1Ge[420, 1] := -7.76796E-02;
aff1Ge[421, 0] := 4.21158E+03; aff1Ge[421, 1] := -8.04621E-02;
aff1Ge[422, 0] := 4.22156E+03; aff1Ge[422, 1] := -8.32471E-02;
aff1Ge[423, 0] := 4.23154E+03; aff1Ge[423, 1] := -8.60343E-02;
aff1Ge[424, 0] := 4.24152E+03; aff1Ge[424, 1] := -8.88238E-02;
aff1Ge[425, 0] := 4.25150E+03; aff1Ge[425, 1] := -9.16151E-02;
aff1Ge[426, 0] := 4.26148E+03; aff1Ge[426, 1] := -9.44083E-02;
aff1Ge[427, 0] := 4.27146E+03; aff1Ge[427, 1] := -9.72031E-02;
aff1Ge[428, 0] := 4.28144E+03; aff1Ge[428, 1] := -9.99993E-02;
aff1Ge[429, 0] := 4.29142E+03; aff1Ge[429, 1] := -1.02797E-01;
aff1Ge[430, 0] := 4.30140E+03; aff1Ge[430, 1] := -1.05596E-01;
aff1Ge[431, 0] := 4.31138E+03; aff1Ge[431, 1] := -1.08395E-01;
aff1Ge[432, 0] := 4.32136E+03; aff1Ge[432, 1] := -1.11196E-01;
aff1Ge[433, 0] := 4.33134E+03; aff1Ge[433, 1] := -1.13997E-01;
aff1Ge[434, 0] := 4.34132E+03; aff1Ge[434, 1] := -1.16799E-01;
aff1Ge[435, 0] := 4.35130E+03; aff1Ge[435, 1] := -1.19601E-01;
aff1Ge[436, 0] := 4.36128E+03; aff1Ge[436, 1] := -1.22403E-01;
aff1Ge[437, 0] := 4.37126E+03; aff1Ge[437, 1] := -1.25206E-01;
aff1Ge[438, 0] := 4.38124E+03; aff1Ge[438, 1] := -1.28009E-01;
aff1Ge[439, 0] := 4.39122E+03; aff1Ge[439, 1] := -1.30811E-01;
aff1Ge[440, 0] := 4.40120E+03; aff1Ge[440, 1] := -1.33614E-01;
aff1Ge[441, 0] := 4.41118E+03; aff1Ge[441, 1] := -1.36416E-01;
aff1Ge[442, 0] := 4.42116E+03; aff1Ge[442, 1] := -1.39217E-01;
aff1Ge[443, 0] := 4.43114E+03; aff1Ge[443, 1] := -1.42018E-01;
aff1Ge[444, 0] := 4.44112E+03; aff1Ge[444, 1] := -1.44818E-01;
aff1Ge[445, 0] := 4.45110E+03; aff1Ge[445, 1] := -1.47618E-01;
aff1Ge[446, 0] := 4.46108E+03; aff1Ge[446, 1] := -1.50416E-01;
aff1Ge[447, 0] := 4.47106E+03; aff1Ge[447, 1] := -1.53214E-01;
aff1Ge[448, 0] := 4.48104E+03; aff1Ge[448, 1] := -1.56010E-01;
aff1Ge[449, 0] := 4.49102E+03; aff1Ge[449, 1] := -1.58805E-01;
aff1Ge[450, 0] := 4.50100E+03; aff1Ge[450, 1] := -1.61599E-01;
aff1Ge[451, 0] := 4.51098E+03; aff1Ge[451, 1] := -1.64392E-01;
aff1Ge[452, 0] := 4.52096E+03; aff1Ge[452, 1] := -1.67183E-01;
aff1Ge[453, 0] := 4.53094E+03; aff1Ge[453, 1] := -1.69972E-01;
aff1Ge[454, 0] := 4.54092E+03; aff1Ge[454, 1] := -1.72760E-01;
aff1Ge[455, 0] := 4.55090E+03; aff1Ge[455, 1] := -1.75545E-01;
aff1Ge[456, 0] := 4.56088E+03; aff1Ge[456, 1] := -1.78329E-01;
aff1Ge[457, 0] := 4.57086E+03; aff1Ge[457, 1] := -1.81112E-01;
aff1Ge[458, 0] := 4.58084E+03; aff1Ge[458, 1] := -1.83892E-01;
aff1Ge[459, 0] := 4.59082E+03; aff1Ge[459, 1] := -1.86670E-01;
aff1Ge[460, 0] := 4.60080E+03; aff1Ge[460, 1] := -1.89445E-01;
aff1Ge[461, 0] := 4.61078E+03; aff1Ge[461, 1] := -1.92219E-01;
aff1Ge[462, 0] := 4.62076E+03; aff1Ge[462, 1] := -1.94990E-01;
aff1Ge[463, 0] := 4.63074E+03; aff1Ge[463, 1] := -1.97759E-01;
aff1Ge[464, 0] := 4.64072E+03; aff1Ge[464, 1] := -2.00525E-01;
aff1Ge[465, 0] := 4.65070E+03; aff1Ge[465, 1] := -2.03289E-01;
aff1Ge[466, 0] := 4.66068E+03; aff1Ge[466, 1] := -2.06050E-01;
aff1Ge[467, 0] := 4.67066E+03; aff1Ge[467, 1] := -2.08808E-01;
aff1Ge[468, 0] := 4.68064E+03; aff1Ge[468, 1] := -2.11564E-01;
aff1Ge[469, 0] := 4.69062E+03; aff1Ge[469, 1] := -2.14316E-01;
aff1Ge[470, 0] := 4.70060E+03; aff1Ge[470, 1] := -2.17066E-01;
aff1Ge[471, 0] := 4.71058E+03; aff1Ge[471, 1] := -2.19813E-01;
aff1Ge[472, 0] := 4.72056E+03; aff1Ge[472, 1] := -2.22557E-01;
aff1Ge[473, 0] := 4.73054E+03; aff1Ge[473, 1] := -2.25298E-01;
aff1Ge[474, 0] := 4.74052E+03; aff1Ge[474, 1] := -2.28035E-01;
aff1Ge[475, 0] := 4.75050E+03; aff1Ge[475, 1] := -2.30770E-01;
aff1Ge[476, 0] := 4.76048E+03; aff1Ge[476, 1] := -2.33501E-01;
aff1Ge[477, 0] := 4.77046E+03; aff1Ge[477, 1] := -2.36229E-01;
aff1Ge[478, 0] := 4.78044E+03; aff1Ge[478, 1] := -2.38953E-01;
aff1Ge[479, 0] := 4.79042E+03; aff1Ge[479, 1] := -2.41674E-01;
aff1Ge[480, 0] := 4.80040E+03; aff1Ge[480, 1] := -2.44392E-01;
aff1Ge[481, 0] := 4.81038E+03; aff1Ge[481, 1] := -2.47106E-01;
aff1Ge[482, 0] := 4.82036E+03; aff1Ge[482, 1] := -2.49816E-01;
aff1Ge[483, 0] := 4.83034E+03; aff1Ge[483, 1] := -2.52523E-01;
aff1Ge[484, 0] := 4.84032E+03; aff1Ge[484, 1] := -2.55226E-01;
aff1Ge[485, 0] := 4.85030E+03; aff1Ge[485, 1] := -2.57926E-01;
aff1Ge[486, 0] := 4.86028E+03; aff1Ge[486, 1] := -2.60621E-01;
aff1Ge[487, 0] := 4.87026E+03; aff1Ge[487, 1] := -2.63313E-01;
aff1Ge[488, 0] := 4.88024E+03; aff1Ge[488, 1] := -2.66001E-01;
aff1Ge[489, 0] := 4.89022E+03; aff1Ge[489, 1] := -2.68685E-01;
aff1Ge[490, 0] := 4.90020E+03; aff1Ge[490, 1] := -2.71365E-01;
aff1Ge[491, 0] := 4.91018E+03; aff1Ge[491, 1] := -2.74041E-01;
aff1Ge[492, 0] := 4.92016E+03; aff1Ge[492, 1] := -2.76712E-01;
aff1Ge[493, 0] := 4.93014E+03; aff1Ge[493, 1] := -2.79380E-01;
aff1Ge[494, 0] := 4.94012E+03; aff1Ge[494, 1] := -2.82043E-01;
aff1Ge[495, 0] := 4.95010E+03; aff1Ge[495, 1] := -2.84702E-01;
aff1Ge[496, 0] := 4.96008E+03; aff1Ge[496, 1] := -2.87357E-01;
aff1Ge[497, 0] := 4.97006E+03; aff1Ge[497, 1] := -2.90008E-01;
aff1Ge[498, 0] := 4.98004E+03; aff1Ge[498, 1] := -2.92654E-01;
aff1Ge[499, 0] := 4.99002E+03; aff1Ge[499, 1] := -2.95296E-01;
aff1Ge[500, 0] := 5.00000E+03; aff1Ge[500, 1] := -2.97933E-01;
aff1Ge[501, 0] := 5.05000E+03; aff1Ge[501, 1] := -3.11077E-01;
aff1Ge[502, 0] := 5.10000E+03; aff1Ge[502, 1] := -3.24102E-01;
aff1Ge[503, 0] := 5.15000E+03; aff1Ge[503, 1] := -3.37002E-01;
aff1Ge[504, 0] := 5.20000E+03; aff1Ge[504, 1] := -3.49769E-01;
aff1Ge[505, 0] := 5.25000E+03; aff1Ge[505, 1] := -3.62398E-01;
aff1Ge[506, 0] := 5.30000E+03; aff1Ge[506, 1] := -3.74887E-01;
aff1Ge[507, 0] := 5.35000E+03; aff1Ge[507, 1] := -3.87376E-01;
aff1Ge[508, 0] := 5.40000E+03; aff1Ge[508, 1] := -3.99884E-01;
aff1Ge[509, 0] := 5.45000E+03; aff1Ge[509, 1] := -4.12417E-01;
aff1Ge[510, 0] := 5.50000E+03; aff1Ge[510, 1] := -4.25006E-01;
aff1Ge[511, 0] := 5.55000E+03; aff1Ge[511, 1] := -4.37674E-01;
aff1Ge[512, 0] := 5.60000E+03; aff1Ge[512, 1] := -4.50378E-01;
aff1Ge[513, 0] := 5.65000E+03; aff1Ge[513, 1] := -4.63073E-01;
aff1Ge[514, 0] := 5.70000E+03; aff1Ge[514, 1] := -4.75778E-01;
aff1Ge[515, 0] := 5.75000E+03; aff1Ge[515, 1] := -4.88478E-01;
aff1Ge[516, 0] := 5.80000E+03; aff1Ge[516, 1] := -5.01163E-01;
aff1Ge[517, 0] := 5.85000E+03; aff1Ge[517, 1] := -5.13826E-01;
aff1Ge[518, 0] := 5.90000E+03; aff1Ge[518, 1] := -5.26465E-01;
aff1Ge[519, 0] := 5.95000E+03; aff1Ge[519, 1] := -5.39045E-01;
aff1Ge[520, 0] := 6.00000E+03; aff1Ge[520, 1] := -5.51579E-01;
aff1Ge[521, 0] := 6.05000E+03; aff1Ge[521, 1] := -5.64099E-01;
aff1Ge[522, 0] := 6.10000E+03; aff1Ge[522, 1] := -5.76565E-01;
aff1Ge[523, 0] := 6.15000E+03; aff1Ge[523, 1] := -5.88974E-01;
aff1Ge[524, 0] := 6.20000E+03; aff1Ge[524, 1] := -6.01417E-01;
aff1Ge[525, 0] := 6.25000E+03; aff1Ge[525, 1] := -6.13927E-01;
aff1Ge[526, 0] := 6.30000E+03; aff1Ge[526, 1] := -6.26494E-01;
aff1Ge[527, 0] := 6.35000E+03; aff1Ge[527, 1] := -6.39110E-01;
aff1Ge[528, 0] := 6.40000E+03; aff1Ge[528, 1] := -6.51769E-01;
aff1Ge[529, 0] := 6.45000E+03; aff1Ge[529, 1] := -6.64468E-01;
aff1Ge[530, 0] := 6.50000E+03; aff1Ge[530, 1] := -6.77203E-01;
aff1Ge[531, 0] := 6.55000E+03; aff1Ge[531, 1] := -6.89971E-01;
aff1Ge[532, 0] := 6.60000E+03; aff1Ge[532, 1] := -7.02771E-01;
aff1Ge[533, 0] := 6.65000E+03; aff1Ge[533, 1] := -7.15601E-01;
aff1Ge[534, 0] := 6.70000E+03; aff1Ge[534, 1] := -7.28462E-01;
aff1Ge[535, 0] := 6.75000E+03; aff1Ge[535, 1] := -7.41354E-01;
aff1Ge[536, 0] := 6.80000E+03; aff1Ge[536, 1] := -7.54276E-01;
aff1Ge[537, 0] := 6.85000E+03; aff1Ge[537, 1] := -7.67231E-01;
aff1Ge[538, 0] := 6.90000E+03; aff1Ge[538, 1] := -7.80219E-01;
aff1Ge[539, 0] := 6.95000E+03; aff1Ge[539, 1] := -7.93242E-01;
aff1Ge[540, 0] := 7.00000E+03; aff1Ge[540, 1] := -8.06303E-01;
aff1Ge[541, 0] := 7.05000E+03; aff1Ge[541, 1] := -8.19404E-01;
aff1Ge[542, 0] := 7.10000E+03; aff1Ge[542, 1] := -8.32547E-01;
aff1Ge[543, 0] := 7.15000E+03; aff1Ge[543, 1] := -8.45736E-01;
aff1Ge[544, 0] := 7.20000E+03; aff1Ge[544, 1] := -8.58973E-01;
aff1Ge[545, 0] := 7.25000E+03; aff1Ge[545, 1] := -8.72261E-01;
aff1Ge[546, 0] := 7.30000E+03; aff1Ge[546, 1] := -8.85605E-01;
aff1Ge[547, 0] := 7.35000E+03; aff1Ge[547, 1] := -8.99009E-01;
aff1Ge[548, 0] := 7.40000E+03; aff1Ge[548, 1] := -9.12476E-01;
aff1Ge[549, 0] := 7.45000E+03; aff1Ge[549, 1] := -9.26010E-01;
aff1Ge[550, 0] := 7.50000E+03; aff1Ge[550, 1] := -9.39617E-01;
aff1Ge[551, 0] := 7.55000E+03; aff1Ge[551, 1] := -9.53301E-01;
aff1Ge[552, 0] := 7.60000E+03; aff1Ge[552, 1] := -9.67066E-01;
aff1Ge[553, 0] := 7.65000E+03; aff1Ge[553, 1] := -9.80919E-01;
aff1Ge[554, 0] := 7.70000E+03; aff1Ge[554, 1] := -9.94864E-01;
aff1Ge[555, 0] := 7.75000E+03; aff1Ge[555, 1] := -1.00891E+00;
aff1Ge[556, 0] := 7.80000E+03; aff1Ge[556, 1] := -1.02306E+00;
aff1Ge[557, 0] := 7.85000E+03; aff1Ge[557, 1] := -1.03731E+00;
aff1Ge[558, 0] := 7.90000E+03; aff1Ge[558, 1] := -1.05169E+00;
aff1Ge[559, 0] := 7.95000E+03; aff1Ge[559, 1] := -1.06619E+00;
aff1Ge[560, 0] := 8.00000E+03; aff1Ge[560, 1] := -1.08082E+00;
aff1Ge[561, 0] := 8.05000E+03; aff1Ge[561, 1] := -1.09558E+00;
aff1Ge[562, 0] := 8.10000E+03; aff1Ge[562, 1] := -1.11050E+00;
aff1Ge[563, 0] := 8.15000E+03; aff1Ge[563, 1] := -1.12556E+00;
aff1Ge[564, 0] := 8.20000E+03; aff1Ge[564, 1] := -1.14079E+00;
aff1Ge[565, 0] := 8.25000E+03; aff1Ge[565, 1] := -1.15619E+00;
aff1Ge[566, 0] := 8.30000E+03; aff1Ge[566, 1] := -1.17177E+00;
aff1Ge[567, 0] := 8.35000E+03; aff1Ge[567, 1] := -1.18754E+00;
aff1Ge[568, 0] := 8.40000E+03; aff1Ge[568, 1] := -1.20351E+00;
aff1Ge[569, 0] := 8.45000E+03; aff1Ge[569, 1] := -1.21969E+00;
aff1Ge[570, 0] := 8.50000E+03; aff1Ge[570, 1] := -1.23610E+00;
aff1Ge[571, 0] := 8.55000E+03; aff1Ge[571, 1] := -1.25273E+00;
aff1Ge[572, 0] := 8.60000E+03; aff1Ge[572, 1] := -1.26961E+00;
aff1Ge[573, 0] := 8.65000E+03; aff1Ge[573, 1] := -1.28675E+00;
aff1Ge[574, 0] := 8.70000E+03; aff1Ge[574, 1] := -1.30416E+00;
aff1Ge[575, 0] := 8.75000E+03; aff1Ge[575, 1] := -1.32186E+00;
aff1Ge[576, 0] := 8.80000E+03; aff1Ge[576, 1] := -1.33985E+00;
aff1Ge[577, 0] := 8.85000E+03; aff1Ge[577, 1] := -1.35815E+00;
aff1Ge[578, 0] := 8.90000E+03; aff1Ge[578, 1] := -1.37679E+00;
aff1Ge[579, 0] := 8.95000E+03; aff1Ge[579, 1] := -1.39585E+00;
aff1Ge[580, 0] := 9.00000E+03; aff1Ge[580, 1] := -1.41541E+00;
aff1Ge[581, 0] := 9.05000E+03; aff1Ge[581, 1] := -1.43553E+00;
aff1Ge[582, 0] := 9.10000E+03; aff1Ge[582, 1] := -1.45622E+00;
aff1Ge[583, 0] := 9.15000E+03; aff1Ge[583, 1] := -1.47747E+00;
aff1Ge[584, 0] := 9.20000E+03; aff1Ge[584, 1] := -1.49932E+00;
aff1Ge[585, 0] := 9.25000E+03; aff1Ge[585, 1] := -1.52178E+00;
aff1Ge[586, 0] := 9.30000E+03; aff1Ge[586, 1] := -1.54490E+00;
aff1Ge[587, 0] := 9.35000E+03; aff1Ge[587, 1] := -1.56870E+00;
aff1Ge[588, 0] := 9.40000E+03; aff1Ge[588, 1] := -1.59322E+00;
aff1Ge[589, 0] := 9.45000E+03; aff1Ge[589, 1] := -1.61851E+00;
aff1Ge[590, 0] := 9.50000E+03; aff1Ge[590, 1] := -1.64461E+00;
aff1Ge[591, 0] := 9.55000E+03; aff1Ge[591, 1] := -1.67158E+00;
aff1Ge[592, 0] := 9.60000E+03; aff1Ge[592, 1] := -1.69948E+00;
aff1Ge[593, 0] := 9.65000E+03; aff1Ge[593, 1] := -1.72837E+00;
aff1Ge[594, 0] := 9.70000E+03; aff1Ge[594, 1] := -1.75833E+00;
aff1Ge[595, 0] := 9.75000E+03; aff1Ge[595, 1] := -1.78944E+00;
aff1Ge[596, 0] := 9.80000E+03; aff1Ge[596, 1] := -1.82179E+00;
aff1Ge[597, 0] := 9.85000E+03; aff1Ge[597, 1] := -1.85548E+00;
aff1Ge[598, 0] := 9.90000E+03; aff1Ge[598, 1] := -1.89064E+00;
aff1Ge[599, 0] := 9.95000E+03; aff1Ge[599, 1] := -1.92740E+00;
aff1Ge[600, 0] := 1.00000E+04; aff1Ge[600, 1] := -1.96590E+00;
aff1Ge[601, 0] := 1.00500E+04; aff1Ge[601, 1] := -2.00631E+00;
aff1Ge[602, 0] := 1.01000E+04; aff1Ge[602, 1] := -2.04885E+00;
aff1Ge[603, 0] := 1.01500E+04; aff1Ge[603, 1] := -2.09373E+00;
aff1Ge[604, 0] := 1.02000E+04; aff1Ge[604, 1] := -2.14123E+00;
aff1Ge[605, 0] := 1.02500E+04; aff1Ge[605, 1] := -2.19165E+00;
aff1Ge[606, 0] := 1.03000E+04; aff1Ge[606, 1] := -2.24538E+00;
aff1Ge[607, 0] := 1.03500E+04; aff1Ge[607, 1] := -2.30286E+00;
aff1Ge[608, 0] := 1.04000E+04; aff1Ge[608, 1] := -2.36463E+00;
aff1Ge[609, 0] := 1.04500E+04; aff1Ge[609, 1] := -2.43135E+00;
aff1Ge[610, 0] := 1.05000E+04; aff1Ge[610, 1] := -2.50387E+00;
aff1Ge[611, 0] := 1.05500E+04; aff1Ge[611, 1] := -2.58316E+00;
aff1Ge[612, 0] := 1.06000E+04; aff1Ge[612, 1] := -2.67074E+00;
aff1Ge[613, 0] := 1.06500E+04; aff1Ge[613, 1] := -2.76810E+00;
aff1Ge[614, 0] := 1.07000E+04; aff1Ge[614, 1] := -2.87831E+00;
aff1Ge[615, 0] := 1.07500E+04; aff1Ge[615, 1] := -3.00367E+00;
aff1Ge[616, 0] := 1.08000E+04; aff1Ge[616, 1] := -3.15215E+00;
aff1Ge[617, 0] := 1.08500E+04; aff1Ge[617, 1] := -3.32695E+00;
aff1Ge[618, 0] := 1.09000E+04; aff1Ge[618, 1] := -3.54568E+00;
aff1Ge[619, 0] := 1.09500E+04; aff1Ge[619, 1] := -3.83175E+00;
aff1Ge[620, 0] := 1.10000E+04; aff1Ge[620, 1] := -4.22308E+00;
aff1Ge[621, 0] := 1.10500E+04; aff1Ge[621, 1] := -4.90280E+00;
aff1Ge[622, 0] := 1.11000E+04; aff1Ge[622, 1] := -7.91070E+00;
aff1Ge[623, 0] := 1.11500E+04; aff1Ge[623, 1] := -4.99587E+00;
aff1Ge[624, 0] := 1.12000E+04; aff1Ge[624, 1] := -4.19048E+00;
aff1Ge[625, 0] := 1.12500E+04; aff1Ge[625, 1] := -3.70028E+00;
aff1Ge[626, 0] := 1.13000E+04; aff1Ge[626, 1] := -3.37927E+00;
aff1Ge[627, 0] := 1.13500E+04; aff1Ge[627, 1] := -3.12255E+00;
aff1Ge[628, 0] := 1.14000E+04; aff1Ge[628, 1] := -2.90829E+00;
aff1Ge[629, 0] := 1.14500E+04; aff1Ge[629, 1] := -2.72625E+00;
aff1Ge[630, 0] := 1.15000E+04; aff1Ge[630, 1] := -2.57094E+00;
aff1Ge[631, 0] := 1.15500E+04; aff1Ge[631, 1] := -2.43566E+00;
aff1Ge[632, 0] := 1.16000E+04; aff1Ge[632, 1] := -2.31492E+00;
aff1Ge[633, 0] := 1.16500E+04; aff1Ge[633, 1] := -2.20724E+00;
aff1Ge[634, 0] := 1.17000E+04; aff1Ge[634, 1] := -2.10939E+00;
aff1Ge[635, 0] := 1.17500E+04; aff1Ge[635, 1] := -2.01993E+00;
aff1Ge[636, 0] := 1.18000E+04; aff1Ge[636, 1] := -1.93704E+00;
aff1Ge[637, 0] := 1.18500E+04; aff1Ge[637, 1] := -1.85980E+00;
aff1Ge[638, 0] := 1.19000E+04; aff1Ge[638, 1] := -1.78771E+00;
aff1Ge[639, 0] := 1.19500E+04; aff1Ge[639, 1] := -1.72029E+00;
aff1Ge[640, 0] := 1.20000E+04; aff1Ge[640, 1] := -1.65704E+00;
aff1Ge[641, 0] := 1.20500E+04; aff1Ge[641, 1] := -1.59745E+00;
aff1Ge[642, 0] := 1.21000E+04; aff1Ge[642, 1] := -1.54118E+00;
aff1Ge[643, 0] := 1.21500E+04; aff1Ge[643, 1] := -1.48792E+00;
aff1Ge[644, 0] := 1.22000E+04; aff1Ge[644, 1] := -1.43739E+00;
aff1Ge[645, 0] := 1.22500E+04; aff1Ge[645, 1] := -1.38937E+00;
aff1Ge[646, 0] := 1.23000E+04; aff1Ge[646, 1] := -1.34363E+00;
aff1Ge[647, 0] := 1.23500E+04; aff1Ge[647, 1] := -1.30000E+00;
aff1Ge[648, 0] := 1.24000E+04; aff1Ge[648, 1] := -1.25830E+00;
aff1Ge[649, 0] := 1.24500E+04; aff1Ge[649, 1] := -1.21840E+00;
aff1Ge[650, 0] := 1.25000E+04; aff1Ge[650, 1] := -1.18016E+00;
aff1Ge[651, 0] := 1.25500E+04; aff1Ge[651, 1] := -1.14347E+00;
aff1Ge[652, 0] := 1.26000E+04; aff1Ge[652, 1] := -1.10821E+00;
aff1Ge[653, 0] := 1.26500E+04; aff1Ge[653, 1] := -1.07430E+00;
aff1Ge[654, 0] := 1.27000E+04; aff1Ge[654, 1] := -1.04165E+00;
aff1Ge[655, 0] := 1.27500E+04; aff1Ge[655, 1] := -1.01017E+00;
aff1Ge[656, 0] := 1.28000E+04; aff1Ge[656, 1] := -9.79805E-01;
aff1Ge[657, 0] := 1.28500E+04; aff1Ge[657, 1] := -9.50477E-01;
aff1Ge[658, 0] := 1.29000E+04; aff1Ge[658, 1] := -9.22128E-01;
aff1Ge[659, 0] := 1.29500E+04; aff1Ge[659, 1] := -8.94703E-01;
aff1Ge[660, 0] := 1.30000E+04; aff1Ge[660, 1] := -8.68152E-01;
aff1Ge[661, 0] := 1.30500E+04; aff1Ge[661, 1] := -8.42426E-01;
aff1Ge[662, 0] := 1.31000E+04; aff1Ge[662, 1] := -8.17483E-01;
aff1Ge[663, 0] := 1.31500E+04; aff1Ge[663, 1] := -7.93281E-01;
aff1Ge[664, 0] := 1.32000E+04; aff1Ge[664, 1] := -7.69782E-01;
aff1Ge[665, 0] := 1.32500E+04; aff1Ge[665, 1] := -7.46953E-01;
aff1Ge[666, 0] := 1.33000E+04; aff1Ge[666, 1] := -7.24759E-01;
aff1Ge[667, 0] := 1.33500E+04; aff1Ge[667, 1] := -7.03171E-01;
aff1Ge[668, 0] := 1.34000E+04; aff1Ge[668, 1] := -6.82161E-01;
aff1Ge[669, 0] := 1.34500E+04; aff1Ge[669, 1] := -6.61700E-01;
aff1Ge[670, 0] := 1.35000E+04; aff1Ge[670, 1] := -6.41764E-01;
aff1Ge[671, 0] := 1.35500E+04; aff1Ge[671, 1] := -6.22329E-01;
aff1Ge[672, 0] := 1.36000E+04; aff1Ge[672, 1] := -6.03374E-01;
aff1Ge[673, 0] := 1.36500E+04; aff1Ge[673, 1] := -5.84875E-01;
aff1Ge[674, 0] := 1.37000E+04; aff1Ge[674, 1] := -5.66814E-01;
aff1Ge[675, 0] := 1.37500E+04; aff1Ge[675, 1] := -5.49172E-01;
aff1Ge[676, 0] := 1.38000E+04; aff1Ge[676, 1] := -5.31929E-01;
aff1Ge[677, 0] := 1.38500E+04; aff1Ge[677, 1] := -5.15068E-01;
aff1Ge[678, 0] := 1.39000E+04; aff1Ge[678, 1] := -4.98573E-01;
aff1Ge[679, 0] := 1.39500E+04; aff1Ge[679, 1] := -4.82426E-01;
aff1Ge[680, 0] := 1.40000E+04; aff1Ge[680, 1] := -4.66611E-01;
aff1Ge[681, 0] := 1.40500E+04; aff1Ge[681, 1] := -4.51112E-01;
aff1Ge[682, 0] := 1.41000E+04; aff1Ge[682, 1] := -4.35915E-01;
aff1Ge[683, 0] := 1.41500E+04; aff1Ge[683, 1] := -4.21002E-01;
aff1Ge[684, 0] := 1.42000E+04; aff1Ge[684, 1] := -4.06351E-01;
aff1Ge[685, 0] := 1.42500E+04; aff1Ge[685, 1] := -3.91947E-01;
aff1Ge[686, 0] := 1.43000E+04; aff1Ge[686, 1] := -3.77774E-01;
aff1Ge[687, 0] := 1.43500E+04; aff1Ge[687, 1] := -3.63808E-01;
aff1Ge[688, 0] := 1.44000E+04; aff1Ge[688, 1] := -3.50020E-01;
aff1Ge[689, 0] := 1.44500E+04; aff1Ge[689, 1] := -3.36462E-01;
aff1Ge[690, 0] := 1.45000E+04; aff1Ge[690, 1] := -3.23219E-01;
aff1Ge[691, 0] := 1.45500E+04; aff1Ge[691, 1] := -3.10365E-01;
aff1Ge[692, 0] := 1.46000E+04; aff1Ge[692, 1] := -2.97885E-01;
aff1Ge[693, 0] := 1.46500E+04; aff1Ge[693, 1] := -2.85739E-01;
aff1Ge[694, 0] := 1.47000E+04; aff1Ge[694, 1] := -2.73893E-01;
aff1Ge[695, 0] := 1.47500E+04; aff1Ge[695, 1] := -2.62337E-01;
aff1Ge[696, 0] := 1.48000E+04; aff1Ge[696, 1] := -2.51061E-01;
aff1Ge[697, 0] := 1.48500E+04; aff1Ge[697, 1] := -2.40056E-01;
aff1Ge[698, 0] := 1.49000E+04; aff1Ge[698, 1] := -2.29310E-01;
aff1Ge[699, 0] := 1.49500E+04; aff1Ge[699, 1] := -2.18813E-01;
aff1Ge[700, 0] := 1.50000E+04; aff1Ge[700, 1] := -2.08556E-01;
aff1Ge[701, 0] := 1.50500E+04; aff1Ge[701, 1] := -1.98532E-01;
aff1Ge[702, 0] := 1.51000E+04; aff1Ge[702, 1] := -1.88732E-01;
aff1Ge[703, 0] := 1.51500E+04; aff1Ge[703, 1] := -1.79151E-01;
aff1Ge[704, 0] := 1.52000E+04; aff1Ge[704, 1] := -1.69780E-01;
aff1Ge[705, 0] := 1.52500E+04; aff1Ge[705, 1] := -1.60614E-01;
aff1Ge[706, 0] := 1.53000E+04; aff1Ge[706, 1] := -1.51647E-01;
aff1Ge[707, 0] := 1.53500E+04; aff1Ge[707, 1] := -1.42874E-01;
aff1Ge[708, 0] := 1.54000E+04; aff1Ge[708, 1] := -1.34288E-01;
aff1Ge[709, 0] := 1.54500E+04; aff1Ge[709, 1] := -1.25886E-01;
aff1Ge[710, 0] := 1.55000E+04; aff1Ge[710, 1] := -1.17661E-01;
aff1Ge[711, 0] := 1.55500E+04; aff1Ge[711, 1] := -1.09611E-01;
aff1Ge[712, 0] := 1.56000E+04; aff1Ge[712, 1] := -1.01729E-01;
aff1Ge[713, 0] := 1.56500E+04; aff1Ge[713, 1] := -9.40117E-02;
aff1Ge[714, 0] := 1.57000E+04; aff1Ge[714, 1] := -8.64555E-02;
aff1Ge[715, 0] := 1.57500E+04; aff1Ge[715, 1] := -7.90559E-02;
aff1Ge[716, 0] := 1.58000E+04; aff1Ge[716, 1] := -7.18093E-02;
aff1Ge[717, 0] := 1.58500E+04; aff1Ge[717, 1] := -6.47120E-02;
aff1Ge[718, 0] := 1.59000E+04; aff1Ge[718, 1] := -5.77602E-02;
aff1Ge[719, 0] := 1.59500E+04; aff1Ge[719, 1] := -5.09507E-02;
aff1Ge[720, 0] := 1.60000E+04; aff1Ge[720, 1] := -4.42803E-02;
aff1Ge[721, 0] := 1.60500E+04; aff1Ge[721, 1] := -3.77456E-02;
aff1Ge[722, 0] := 1.61000E+04; aff1Ge[722, 1] := -3.13436E-02;
aff1Ge[723, 0] := 1.61500E+04; aff1Ge[723, 1] := -2.50713E-02;
aff1Ge[724, 0] := 1.62000E+04; aff1Ge[724, 1] := -1.89258E-02;
aff1Ge[725, 0] := 1.62500E+04; aff1Ge[725, 1] := -1.29042E-02;
aff1Ge[726, 0] := 1.63000E+04; aff1Ge[726, 1] := -7.00377E-03;
aff1Ge[727, 0] := 1.63500E+04; aff1Ge[727, 1] := -1.22192E-03;
aff1Ge[728, 0] := 1.64000E+04; aff1Ge[728, 1] := 4.44395E-03;
aff1Ge[729, 0] := 1.64500E+04; aff1Ge[729, 1] := 9.99634E-03;
aff1Ge[730, 0] := 1.65000E+04; aff1Ge[730, 1] := 1.54377E-02;
aff1Ge[731, 0] := 1.65500E+04; aff1Ge[731, 1] := 2.07704E-02;
aff1Ge[732, 0] := 1.66000E+04; aff1Ge[732, 1] := 2.59967E-02;
aff1Ge[733, 0] := 1.66500E+04; aff1Ge[733, 1] := 3.11192E-02;
aff1Ge[734, 0] := 1.67000E+04; aff1Ge[734, 1] := 3.61404E-02;
aff1Ge[735, 0] := 1.67500E+04; aff1Ge[735, 1] := 4.10621E-02;
aff1Ge[736, 0] := 1.68000E+04; aff1Ge[736, 1] := 4.58851E-02;
aff1Ge[737, 0] := 1.68500E+04; aff1Ge[737, 1] := 5.06100E-02;
aff1Ge[738, 0] := 1.69000E+04; aff1Ge[738, 1] := 5.52383E-02;
aff1Ge[739, 0] := 1.69500E+04; aff1Ge[739, 1] := 5.97737E-02;
aff1Ge[740, 0] := 1.70000E+04; aff1Ge[740, 1] := 6.42204E-02;
aff1Ge[741, 0] := 1.70500E+04; aff1Ge[741, 1] := 6.85822E-02;
aff1Ge[742, 0] := 1.71000E+04; aff1Ge[742, 1] := 7.28602E-02;
aff1Ge[743, 0] := 1.71500E+04; aff1Ge[743, 1] := 7.70548E-02;
aff1Ge[744, 0] := 1.72000E+04; aff1Ge[744, 1] := 8.11663E-02;
aff1Ge[745, 0] := 1.72500E+04; aff1Ge[745, 1] := 8.51959E-02;
aff1Ge[746, 0] := 1.73000E+04; aff1Ge[746, 1] := 8.91454E-02;
aff1Ge[747, 0] := 1.73500E+04; aff1Ge[747, 1] := 9.30169E-02;
aff1Ge[748, 0] := 1.74000E+04; aff1Ge[748, 1] := 9.68122E-02;
aff1Ge[749, 0] := 1.74500E+04; aff1Ge[749, 1] := 1.00533E-01;
aff1Ge[750, 0] := 1.75000E+04; aff1Ge[750, 1] := 1.04180E-01;
aff1Ge[751, 0] := 1.75500E+04; aff1Ge[751, 1] := 1.07755E-01;
aff1Ge[752, 0] := 1.76000E+04; aff1Ge[752, 1] := 1.11259E-01;
aff1Ge[753, 0] := 1.76500E+04; aff1Ge[753, 1] := 1.14694E-01;
aff1Ge[754, 0] := 1.77000E+04; aff1Ge[754, 1] := 1.18061E-01;
aff1Ge[755, 0] := 1.77500E+04; aff1Ge[755, 1] := 1.21362E-01;
aff1Ge[756, 0] := 1.78000E+04; aff1Ge[756, 1] := 1.24597E-01;
aff1Ge[757, 0] := 1.78500E+04; aff1Ge[757, 1] := 1.27768E-01;
aff1Ge[758, 0] := 1.79000E+04; aff1Ge[758, 1] := 1.30877E-01;
aff1Ge[759, 0] := 1.79500E+04; aff1Ge[759, 1] := 1.33924E-01;
aff1Ge[760, 0] := 1.80000E+04; aff1Ge[760, 1] := 1.36911E-01;
aff1Ge[761, 0] := 1.80500E+04; aff1Ge[761, 1] := 1.39838E-01;
aff1Ge[762, 0] := 1.81000E+04; aff1Ge[762, 1] := 1.42707E-01;
aff1Ge[763, 0] := 1.81500E+04; aff1Ge[763, 1] := 1.45520E-01;
aff1Ge[764, 0] := 1.82000E+04; aff1Ge[764, 1] := 1.48276E-01;
aff1Ge[765, 0] := 1.82500E+04; aff1Ge[765, 1] := 1.50978E-01;
aff1Ge[766, 0] := 1.83000E+04; aff1Ge[766, 1] := 1.53626E-01;
aff1Ge[767, 0] := 1.83500E+04; aff1Ge[767, 1] := 1.56221E-01;
aff1Ge[768, 0] := 1.84000E+04; aff1Ge[768, 1] := 1.58764E-01;
aff1Ge[769, 0] := 1.84500E+04; aff1Ge[769, 1] := 1.61257E-01;
aff1Ge[770, 0] := 1.85000E+04; aff1Ge[770, 1] := 1.63700E-01;
aff1Ge[771, 0] := 1.85500E+04; aff1Ge[771, 1] := 1.66093E-01;
aff1Ge[772, 0] := 1.86000E+04; aff1Ge[772, 1] := 1.68439E-01;
aff1Ge[773, 0] := 1.86500E+04; aff1Ge[773, 1] := 1.70738E-01;
aff1Ge[774, 0] := 1.87000E+04; aff1Ge[774, 1] := 1.72991E-01;
aff1Ge[775, 0] := 1.87500E+04; aff1Ge[775, 1] := 1.75198E-01;
aff1Ge[776, 0] := 1.88000E+04; aff1Ge[776, 1] := 1.77361E-01;
aff1Ge[777, 0] := 1.88500E+04; aff1Ge[777, 1] := 1.79481E-01;
aff1Ge[778, 0] := 1.89000E+04; aff1Ge[778, 1] := 1.81557E-01;
aff1Ge[779, 0] := 1.89500E+04; aff1Ge[779, 1] := 1.83592E-01;
aff1Ge[780, 0] := 1.90000E+04; aff1Ge[780, 1] := 1.85585E-01;
aff1Ge[781, 0] := 1.90500E+04; aff1Ge[781, 1] := 1.87538E-01;
aff1Ge[782, 0] := 1.91000E+04; aff1Ge[782, 1] := 1.89452E-01;
aff1Ge[783, 0] := 1.91500E+04; aff1Ge[783, 1] := 1.91326E-01;
aff1Ge[784, 0] := 1.92000E+04; aff1Ge[784, 1] := 1.93162E-01;
aff1Ge[785, 0] := 1.92500E+04; aff1Ge[785, 1] := 1.94961E-01;
aff1Ge[786, 0] := 1.93000E+04; aff1Ge[786, 1] := 1.96723E-01;
aff1Ge[787, 0] := 1.93500E+04; aff1Ge[787, 1] := 1.98449E-01;
aff1Ge[788, 0] := 1.94000E+04; aff1Ge[788, 1] := 2.00139E-01;
aff1Ge[789, 0] := 1.94500E+04; aff1Ge[789, 1] := 2.01795E-01;
aff1Ge[790, 0] := 1.95000E+04; aff1Ge[790, 1] := 2.03416E-01;
aff1Ge[791, 0] := 1.95500E+04; aff1Ge[791, 1] := 2.05004E-01;
aff1Ge[792, 0] := 1.96000E+04; aff1Ge[792, 1] := 2.06560E-01;
aff1Ge[793, 0] := 1.96500E+04; aff1Ge[793, 1] := 2.08083E-01;
aff1Ge[794, 0] := 1.97000E+04; aff1Ge[794, 1] := 2.09574E-01;
aff1Ge[795, 0] := 1.97500E+04; aff1Ge[795, 1] := 2.11034E-01;
aff1Ge[796, 0] := 1.98000E+04; aff1Ge[796, 1] := 2.12464E-01;
aff1Ge[797, 0] := 1.98500E+04; aff1Ge[797, 1] := 2.13865E-01;
aff1Ge[798, 0] := 1.99000E+04; aff1Ge[798, 1] := 2.15235E-01;
aff1Ge[799, 0] := 1.99500E+04; aff1Ge[799, 1] := 2.16577E-01;
aff1Ge[800, 0] := 2.00000E+04; aff1Ge[800, 1] := 2.17891E-01;
aff1Ge[801, 0] := 2.00500E+04; aff1Ge[801, 1] := 2.19177E-01;
aff1Ge[802, 0] := 2.01000E+04; aff1Ge[802, 1] := 2.20436E-01;
aff1Ge[803, 0] := 2.01500E+04; aff1Ge[803, 1] := 2.21668E-01;
aff1Ge[804, 0] := 2.02000E+04; aff1Ge[804, 1] := 2.22875E-01;
aff1Ge[805, 0] := 2.02500E+04; aff1Ge[805, 1] := 2.24055E-01;
aff1Ge[806, 0] := 2.03000E+04; aff1Ge[806, 1] := 2.25211E-01;
aff1Ge[807, 0] := 2.03500E+04; aff1Ge[807, 1] := 2.26341E-01;
aff1Ge[808, 0] := 2.04000E+04; aff1Ge[808, 1] := 2.27448E-01;
aff1Ge[809, 0] := 2.04500E+04; aff1Ge[809, 1] := 2.28531E-01;
aff1Ge[810, 0] := 2.05000E+04; aff1Ge[810, 1] := 2.29590E-01;
aff1Ge[811, 0] := 2.05500E+04; aff1Ge[811, 1] := 2.30627E-01;
aff1Ge[812, 0] := 2.06000E+04; aff1Ge[812, 1] := 2.31641E-01;
aff1Ge[813, 0] := 2.06500E+04; aff1Ge[813, 1] := 2.32633E-01;
aff1Ge[814, 0] := 2.07000E+04; aff1Ge[814, 1] := 2.33604E-01;
aff1Ge[815, 0] := 2.07500E+04; aff1Ge[815, 1] := 2.34554E-01;
aff1Ge[816, 0] := 2.08000E+04; aff1Ge[816, 1] := 2.35483E-01;
aff1Ge[817, 0] := 2.08500E+04; aff1Ge[817, 1] := 2.36392E-01;
aff1Ge[818, 0] := 2.09000E+04; aff1Ge[818, 1] := 2.37281E-01;
aff1Ge[819, 0] := 2.09500E+04; aff1Ge[819, 1] := 2.38150E-01;
aff1Ge[820, 0] := 2.10000E+04; aff1Ge[820, 1] := 2.39001E-01;
aff1Ge[821, 0] := 2.10500E+04; aff1Ge[821, 1] := 2.39832E-01;
aff1Ge[822, 0] := 2.11000E+04; aff1Ge[822, 1] := 2.40646E-01;
aff1Ge[823, 0] := 2.11500E+04; aff1Ge[823, 1] := 2.41441E-01;
aff1Ge[824, 0] := 2.12000E+04; aff1Ge[824, 1] := 2.42219E-01;
aff1Ge[825, 0] := 2.12500E+04; aff1Ge[825, 1] := 2.42980E-01;
aff1Ge[826, 0] := 2.13000E+04; aff1Ge[826, 1] := 2.43723E-01;
aff1Ge[827, 0] := 2.13500E+04; aff1Ge[827, 1] := 2.44451E-01;
aff1Ge[828, 0] := 2.14000E+04; aff1Ge[828, 1] := 2.45162E-01;
aff1Ge[829, 0] := 2.14500E+04; aff1Ge[829, 1] := 2.45857E-01;
aff1Ge[830, 0] := 2.15000E+04; aff1Ge[830, 1] := 2.46537E-01;
aff1Ge[831, 0] := 2.15500E+04; aff1Ge[831, 1] := 2.47202E-01;
aff1Ge[832, 0] := 2.16000E+04; aff1Ge[832, 1] := 2.47874E-01;
aff1Ge[833, 0] := 2.16500E+04; aff1Ge[833, 1] := 2.48727E-01;
aff1Ge[834, 0] := 2.17000E+04; aff1Ge[834, 1] := 2.49536E-01;
aff1Ge[835, 0] := 2.17500E+04; aff1Ge[835, 1] := 2.50152E-01;
aff1Ge[836, 0] := 2.18000E+04; aff1Ge[836, 1] := 2.50428E-01;
aff1Ge[837, 0] := 2.18500E+04; aff1Ge[837, 1] := 2.49727E-01;
aff1Ge[838, 0] := 2.19000E+04; aff1Ge[838, 1] := 2.48788E-01;
aff1Ge[839, 0] := 2.19500E+04; aff1Ge[839, 1] := 2.48736E-01;
aff1Ge[840, 0] := 2.20000E+04; aff1Ge[840, 1] := 2.50597E-01;
aff1Ge[841, 0] := 2.20500E+04; aff1Ge[841, 1] := 2.55706E-01;
aff1Ge[842, 0] := 2.21000E+04; aff1Ge[842, 1] := 2.64278E-01;
aff1Ge[843, 0] := 2.21500E+04; aff1Ge[843, 1] := 2.74311E-01;
aff1Ge[844, 0] := 2.22000E+04; aff1Ge[844, 1] := 2.84026E-01;
aff1Ge[845, 0] := 2.22500E+04; aff1Ge[845, 1] := 2.91628E-01;
aff1Ge[846, 0] := 2.23000E+04; aff1Ge[846, 1] := 2.95347E-01;
aff1Ge[847, 0] := 2.23500E+04; aff1Ge[847, 1] := 2.96204E-01;
aff1Ge[848, 0] := 2.24000E+04; aff1Ge[848, 1] := 2.95323E-01;
aff1Ge[849, 0] := 2.24500E+04; aff1Ge[849, 1] := 2.93829E-01;
aff1Ge[850, 0] := 2.25000E+04; aff1Ge[850, 1] := 2.92948E-01;
aff1Ge[851, 0] := 2.25500E+04; aff1Ge[851, 1] := 2.92933E-01;
aff1Ge[852, 0] := 2.26000E+04; aff1Ge[852, 1] := 2.93423E-01;
aff1Ge[853, 0] := 2.26500E+04; aff1Ge[853, 1] := 2.94162E-01;
aff1Ge[854, 0] := 2.27000E+04; aff1Ge[854, 1] := 2.94874E-01;
aff1Ge[855, 0] := 2.27500E+04; aff1Ge[855, 1] := 2.95280E-01;
aff1Ge[856, 0] := 2.28000E+04; aff1Ge[856, 1] := 2.95579E-01;
aff1Ge[857, 0] := 2.28500E+04; aff1Ge[857, 1] := 2.95808E-01;
aff1Ge[858, 0] := 2.29000E+04; aff1Ge[858, 1] := 2.96004E-01;
aff1Ge[859, 0] := 2.29500E+04; aff1Ge[859, 1] := 2.96225E-01;
aff1Ge[860, 0] := 2.30000E+04; aff1Ge[860, 1] := 2.96459E-01;
aff1Ge[861, 0] := 2.30500E+04; aff1Ge[861, 1] := 2.96681E-01;
aff1Ge[862, 0] := 2.31000E+04; aff1Ge[862, 1] := 2.96891E-01;
aff1Ge[863, 0] := 2.31500E+04; aff1Ge[863, 1] := 2.97089E-01;
aff1Ge[864, 0] := 2.32000E+04; aff1Ge[864, 1] := 2.97276E-01;
aff1Ge[865, 0] := 2.32500E+04; aff1Ge[865, 1] := 2.97451E-01;
aff1Ge[866, 0] := 2.33000E+04; aff1Ge[866, 1] := 2.97615E-01;
aff1Ge[867, 0] := 2.33500E+04; aff1Ge[867, 1] := 2.97769E-01;
aff1Ge[868, 0] := 2.34000E+04; aff1Ge[868, 1] := 2.97912E-01;
aff1Ge[869, 0] := 2.34500E+04; aff1Ge[869, 1] := 2.98045E-01;
aff1Ge[870, 0] := 2.35000E+04; aff1Ge[870, 1] := 2.98168E-01;
aff1Ge[871, 0] := 2.35500E+04; aff1Ge[871, 1] := 2.98282E-01;
aff1Ge[872, 0] := 2.36000E+04; aff1Ge[872, 1] := 2.98385E-01;
aff1Ge[873, 0] := 2.36500E+04; aff1Ge[873, 1] := 2.98480E-01;
aff1Ge[874, 0] := 2.37000E+04; aff1Ge[874, 1] := 2.98565E-01;
aff1Ge[875, 0] := 2.37500E+04; aff1Ge[875, 1] := 2.98641E-01;
aff1Ge[876, 0] := 2.38000E+04; aff1Ge[876, 1] := 2.98708E-01;
aff1Ge[877, 0] := 2.38500E+04; aff1Ge[877, 1] := 2.98767E-01;
aff1Ge[878, 0] := 2.39000E+04; aff1Ge[878, 1] := 2.98817E-01;
aff1Ge[879, 0] := 2.39500E+04; aff1Ge[879, 1] := 2.98859E-01;
aff1Ge[880, 0] := 2.40000E+04; aff1Ge[880, 1] := 2.98893E-01;
aff1Ge[881, 0] := 2.40500E+04; aff1Ge[881, 1] := 2.98919E-01;
aff1Ge[882, 0] := 2.41000E+04; aff1Ge[882, 1] := 2.98937E-01;
aff1Ge[883, 0] := 2.41500E+04; aff1Ge[883, 1] := 2.98948E-01;
aff1Ge[884, 0] := 2.42000E+04; aff1Ge[884, 1] := 2.98952E-01;
aff1Ge[885, 0] := 2.42500E+04; aff1Ge[885, 1] := 2.98948E-01;
aff1Ge[886, 0] := 2.43000E+04; aff1Ge[886, 1] := 2.98937E-01;
aff1Ge[887, 0] := 2.43500E+04; aff1Ge[887, 1] := 2.98919E-01;
aff1Ge[888, 0] := 2.44000E+04; aff1Ge[888, 1] := 2.98894E-01;
aff1Ge[889, 0] := 2.44500E+04; aff1Ge[889, 1] := 2.98863E-01;
aff1Ge[890, 0] := 2.45000E+04; aff1Ge[890, 1] := 2.98825E-01;
aff1Ge[891, 0] := 2.45500E+04; aff1Ge[891, 1] := 2.98781E-01;
aff1Ge[892, 0] := 2.46000E+04; aff1Ge[892, 1] := 2.98730E-01;
aff1Ge[893, 0] := 2.46500E+04; aff1Ge[893, 1] := 2.98674E-01;
aff1Ge[894, 0] := 2.47000E+04; aff1Ge[894, 1] := 2.98611E-01;
aff1Ge[895, 0] := 2.47500E+04; aff1Ge[895, 1] := 2.98543E-01;
aff1Ge[896, 0] := 2.48000E+04; aff1Ge[896, 1] := 2.98469E-01;
aff1Ge[897, 0] := 2.48500E+04; aff1Ge[897, 1] := 2.98389E-01;
aff1Ge[898, 0] := 2.49000E+04; aff1Ge[898, 1] := 2.98304E-01;
aff1Ge[899, 0] := 2.49500E+04; aff1Ge[899, 1] := 2.98213E-01;
aff1Ge[900, 0] := 2.50000E+04; aff1Ge[900, 1] := 2.98118E-01;
aff1Ge[901, 0] := 2.50500E+04; aff1Ge[901, 1] := 2.98017E-01;
aff1Ge[902, 0] := 2.51000E+04; aff1Ge[902, 1] := 2.97911E-01;
aff1Ge[903, 0] := 2.51500E+04; aff1Ge[903, 1] := 2.97801E-01;
aff1Ge[904, 0] := 2.52000E+04; aff1Ge[904, 1] := 2.97685E-01;
aff1Ge[905, 0] := 2.52500E+04; aff1Ge[905, 1] := 2.97565E-01;
aff1Ge[906, 0] := 2.53000E+04; aff1Ge[906, 1] := 2.97441E-01;
aff1Ge[907, 0] := 2.53500E+04; aff1Ge[907, 1] := 2.97312E-01;
aff1Ge[908, 0] := 2.54000E+04; aff1Ge[908, 1] := 2.97179E-01;
aff1Ge[909, 0] := 2.54500E+04; aff1Ge[909, 1] := 2.97042E-01;
aff1Ge[910, 0] := 2.55000E+04; aff1Ge[910, 1] := 2.96900E-01;
aff1Ge[911, 0] := 2.55500E+04; aff1Ge[911, 1] := 2.96755E-01;
aff1Ge[912, 0] := 2.56000E+04; aff1Ge[912, 1] := 2.96606E-01;
aff1Ge[913, 0] := 2.56500E+04; aff1Ge[913, 1] := 2.96453E-01;
aff1Ge[914, 0] := 2.57000E+04; aff1Ge[914, 1] := 2.96296E-01;
aff1Ge[915, 0] := 2.57500E+04; aff1Ge[915, 1] := 2.96136E-01;
aff1Ge[916, 0] := 2.58000E+04; aff1Ge[916, 1] := 2.95973E-01;
aff1Ge[917, 0] := 2.58500E+04; aff1Ge[917, 1] := 2.95806E-01;
aff1Ge[918, 0] := 2.59000E+04; aff1Ge[918, 1] := 2.95637E-01;
aff1Ge[919, 0] := 2.59500E+04; aff1Ge[919, 1] := 2.95464E-01;
aff1Ge[920, 0] := 2.60000E+04; aff1Ge[920, 1] := 2.95288E-01;
aff1Ge[921, 0] := 2.60500E+04; aff1Ge[921, 1] := 2.95110E-01;
aff1Ge[922, 0] := 2.61000E+04; aff1Ge[922, 1] := 2.94929E-01;
aff1Ge[923, 0] := 2.61500E+04; aff1Ge[923, 1] := 2.94745E-01;
aff1Ge[924, 0] := 2.62000E+04; aff1Ge[924, 1] := 2.94559E-01;
aff1Ge[925, 0] := 2.62500E+04; aff1Ge[925, 1] := 2.94371E-01;
aff1Ge[926, 0] := 2.63000E+04; aff1Ge[926, 1] := 2.94181E-01;
aff1Ge[927, 0] := 2.63500E+04; aff1Ge[927, 1] := 2.93988E-01;
aff1Ge[928, 0] := 2.64000E+04; aff1Ge[928, 1] := 2.93792E-01;
aff1Ge[929, 0] := 2.64500E+04; aff1Ge[929, 1] := 2.93595E-01;
aff1Ge[930, 0] := 2.65000E+04; aff1Ge[930, 1] := 2.93401E-01;
aff1Ge[931, 0] := 2.65500E+04; aff1Ge[931, 1] := 2.93211E-01;
aff1Ge[932, 0] := 2.66000E+04; aff1Ge[932, 1] := 2.93029E-01;
aff1Ge[933, 0] := 2.66500E+04; aff1Ge[933, 1] := 2.92860E-01;
aff1Ge[934, 0] := 2.67000E+04; aff1Ge[934, 1] := 2.92700E-01;
aff1Ge[935, 0] := 2.67500E+04; aff1Ge[935, 1] := 2.92543E-01;
aff1Ge[936, 0] := 2.68000E+04; aff1Ge[936, 1] := 2.92385E-01;
aff1Ge[937, 0] := 2.68500E+04; aff1Ge[937, 1] := 2.92219E-01;
aff1Ge[938, 0] := 2.69000E+04; aff1Ge[938, 1] := 2.92041E-01;
aff1Ge[939, 0] := 2.69500E+04; aff1Ge[939, 1] := 2.91846E-01;
aff1Ge[940, 0] := 2.70000E+04; aff1Ge[940, 1] := 2.91639E-01;
aff1Ge[941, 0] := 2.70500E+04; aff1Ge[941, 1] := 2.91420E-01;
aff1Ge[942, 0] := 2.71000E+04; aff1Ge[942, 1] := 2.91193E-01;
aff1Ge[943, 0] := 2.71500E+04; aff1Ge[943, 1] := 2.90958E-01;
aff1Ge[944, 0] := 2.72000E+04; aff1Ge[944, 1] := 2.90719E-01;
aff1Ge[945, 0] := 2.72500E+04; aff1Ge[945, 1] := 2.90475E-01;
aff1Ge[946, 0] := 2.73000E+04; aff1Ge[946, 1] := 2.90225E-01;
aff1Ge[947, 0] := 2.73500E+04; aff1Ge[947, 1] := 2.89969E-01;
aff1Ge[948, 0] := 2.74000E+04; aff1Ge[948, 1] := 2.89707E-01;
aff1Ge[949, 0] := 2.74500E+04; aff1Ge[949, 1] := 2.89439E-01;
aff1Ge[950, 0] := 2.75000E+04; aff1Ge[950, 1] := 2.89165E-01;
aff1Ge[951, 0] := 2.75500E+04; aff1Ge[951, 1] := 2.88885E-01;
aff1Ge[952, 0] := 2.76000E+04; aff1Ge[952, 1] := 2.88600E-01;
aff1Ge[953, 0] := 2.76500E+04; aff1Ge[953, 1] := 2.88310E-01;
aff1Ge[954, 0] := 2.77000E+04; aff1Ge[954, 1] := 2.88016E-01;
aff1Ge[955, 0] := 2.77500E+04; aff1Ge[955, 1] := 2.87716E-01;
aff1Ge[956, 0] := 2.78000E+04; aff1Ge[956, 1] := 2.87412E-01;
aff1Ge[957, 0] := 2.78500E+04; aff1Ge[957, 1] := 2.87103E-01;
aff1Ge[958, 0] := 2.79000E+04; aff1Ge[958, 1] := 2.86790E-01;
aff1Ge[959, 0] := 2.79500E+04; aff1Ge[959, 1] := 2.86472E-01;
aff1Ge[960, 0] := 2.80000E+04; aff1Ge[960, 1] := 2.86151E-01;
aff1Ge[961, 0] := 2.80500E+04; aff1Ge[961, 1] := 2.85825E-01;
aff1Ge[962, 0] := 2.81000E+04; aff1Ge[962, 1] := 2.85496E-01;
aff1Ge[963, 0] := 2.81500E+04; aff1Ge[963, 1] := 2.85162E-01;
aff1Ge[964, 0] := 2.82000E+04; aff1Ge[964, 1] := 2.84825E-01;
aff1Ge[965, 0] := 2.82500E+04; aff1Ge[965, 1] := 2.84485E-01;
aff1Ge[966, 0] := 2.83000E+04; aff1Ge[966, 1] := 2.84141E-01;
aff1Ge[967, 0] := 2.83500E+04; aff1Ge[967, 1] := 2.83793E-01;
aff1Ge[968, 0] := 2.84000E+04; aff1Ge[968, 1] := 2.83443E-01;
aff1Ge[969, 0] := 2.84500E+04; aff1Ge[969, 1] := 2.83089E-01;
aff1Ge[970, 0] := 2.85000E+04; aff1Ge[970, 1] := 2.82731E-01;
aff1Ge[971, 0] := 2.85500E+04; aff1Ge[971, 1] := 2.82371E-01;
aff1Ge[972, 0] := 2.86000E+04; aff1Ge[972, 1] := 2.82008E-01;
aff1Ge[973, 0] := 2.86500E+04; aff1Ge[973, 1] := 2.81642E-01;
aff1Ge[974, 0] := 2.87000E+04; aff1Ge[974, 1] := 2.81274E-01;
aff1Ge[975, 0] := 2.87500E+04; aff1Ge[975, 1] := 2.80902E-01;
aff1Ge[976, 0] := 2.88000E+04; aff1Ge[976, 1] := 2.80528E-01;
aff1Ge[977, 0] := 2.88500E+04; aff1Ge[977, 1] := 2.80151E-01;
aff1Ge[978, 0] := 2.89000E+04; aff1Ge[978, 1] := 2.79772E-01;
aff1Ge[979, 0] := 2.89500E+04; aff1Ge[979, 1] := 2.79390E-01;
aff1Ge[980, 0] := 2.90000E+04; aff1Ge[980, 1] := 2.79006E-01;
aff1Ge[981, 0] := 2.90500E+04; aff1Ge[981, 1] := 2.78620E-01;
aff1Ge[982, 0] := 2.91000E+04; aff1Ge[982, 1] := 2.78231E-01;
aff1Ge[983, 0] := 2.91500E+04; aff1Ge[983, 1] := 2.77840E-01;
aff1Ge[984, 0] := 2.92000E+04; aff1Ge[984, 1] := 2.77447E-01;
aff1Ge[985, 0] := 2.92500E+04; aff1Ge[985, 1] := 2.77052E-01;
aff1Ge[986, 0] := 2.93000E+04; aff1Ge[986, 1] := 2.76655E-01;
aff1Ge[987, 0] := 2.93500E+04; aff1Ge[987, 1] := 2.76255E-01;
aff1Ge[988, 0] := 2.94000E+04; aff1Ge[988, 1] := 2.75854E-01;
aff1Ge[989, 0] := 2.94500E+04; aff1Ge[989, 1] := 2.75451E-01;
aff1Ge[990, 0] := 2.95000E+04; aff1Ge[990, 1] := 2.75047E-01;
aff1Ge[991, 0] := 2.95500E+04; aff1Ge[991, 1] := 2.74640E-01;
aff1Ge[992, 0] := 2.96000E+04; aff1Ge[992, 1] := 2.74232E-01;
aff1Ge[993, 0] := 2.96500E+04; aff1Ge[993, 1] := 2.73822E-01;
aff1Ge[994, 0] := 2.97000E+04; aff1Ge[994, 1] := 2.73410E-01;
aff1Ge[995, 0] := 2.97500E+04; aff1Ge[995, 1] := 2.72996E-01;
aff1Ge[996, 0] := 2.98000E+04; aff1Ge[996, 1] := 2.72582E-01;
aff1Ge[997, 0] := 2.98500E+04; aff1Ge[997, 1] := 2.72165E-01;
aff1Ge[998, 0] := 2.99000E+04; aff1Ge[998, 1] := 2.71747E-01;
aff1Ge[999, 0] := 2.99500E+04; aff1Ge[999, 1] := 2.71328E-01;

// Element = C

